(* Logix 5000 project; controller Comas_L4 vendor 1 type 14 code 193 rev 30.11; software revision 30.02; part 6 of 12 *)

        [6].Comas.Tete.Cam_Axe_Horizontal_Pan.C.x := 5.0, [6].Comas.Tete.Cam_Axe_Horizontal_Pan.C.y := 2.0, [6].Comas.Tete.Cam_Axe_Horizontal_Pan.D.x := 25.0, [6].Comas.Tete.Cam_Axe_Horizontal_Pan.D.y := 27.0, [6].Comas.Tete.Cam_Axe_Horizontal_Pan.E.x := 10.0, [6].Comas.Tete.Cam_Axe_Horizontal_Pan.E.y := 10.0, [6].Comas.Tete.Cam_Axe_Horizontal_Pan.F.x := 5.0, [6].Comas.Tete.Cam_Axe_Horizontal_Pan.G.x := 10.0, [6].Comas.Tete.Cam_Axe_Horizontal_Pan.G.y := -10.0, [6].Comas.Tete.Cam_Axe_Vertical_Pan.K.x := -10.0, [6].Comas.Tete.Cam_Axe_Vertical_Pan.L.x := -10.0, [6].Comas.Tete.Cam_Axe_Vertical_Pan.L.y := 12.0, [6].Comas.Tete.Cam_Axe_Vertical_Pan.M.x := 5.0, [6].Comas.Tete.Cam_Axe_Vertical_Pan.M.y := 5.0, [6].Comas.Tete.Cam_Axe_Vertical_Pan.N.x := 10.0, [6].Comas.Tete.Offset_Vertical_Droit := 45.0, [6].Comas.Tete.Offset_Horizontal_Droit := 95.0, [6].Comas.Tete.Reserve_Real1 := 3.0, [6].Comas.Pompe.Start_Cam_Logique_Avance := -9.0, [6].Comas.Pompe.Stop_Cam_Logique_Avance := 16.0, [6].Comas.Pompe.Start_Cam_Logique_Recul := 21.0, [6].Comas.Pompe.Stop_Cam_Logique_Recul := 33.0, [6].Comas.Pompe.Consigne_Vitesse_Avance := 19.6, [6].Comas.Pompe.Consigne_Acc_Dec_Avance := 40.0, [6].Comas.Pompe.Consigne_Jerk_Avance := 100.0, [6].Comas.Pompe.Consigne_Vitesse_Recul := -19.0, [6].Comas.Pompe.Consigne_Acc_Dec_Recul := 40.0, [6].Comas.Pompe.Consigne_Jerk_Recul := 100.0, [6].Comas.Pompe.Points_Pan.O.x := -15.0, [6].Comas.Pompe.Points_Pan.Q.x := 25.0, [6].Comas.Pompe.Points_Pan.U.x := 12.0, [6].Comas.Pompe.Reserve_Bool1 := 1, [6].Comas.Rouleaux.Syncho_Pompe := 1, [6].Comas.Rouleaux.Consigne_Vitesse := 25.0, [6].Comas.Rouleaux.Consigne_Acc_Dec := 40.0, [6].Comas.Rouleaux.Consigne_Jerk := 100.0, [6].Comas.Coupe_Fil.Start_Cam_Logique_Virtuelle := 11.0, [6].Comas.Coupe_Fil.Stop_Cam_Logique_Virtuelle := 21.0, [6].Comas.Coupe_Fil.Consigne_Vitesse_Virtuelle := 200.0, [6].Comas.Coupe_Fil.Consigne_Acc_Dec_Virtuelle := 1000.0, [6].Comas.Coupe_Fil.Consigne_Jerk_Virtuelle := 50.0, [6].Comas.Coupe_Fil.Cam_Axe[0].SegmentType := 1, [6].Comas.Coupe_Fil.Cam_Axe[1].Master := 180.0, [6].Comas.Coupe_Fil.Cam_Axe[1].Slave := 90.0, [6].Comas.Coupe_Fil.Cam_Axe[2].Master := 360.0, [6].Comas.Coupe_Fil.Cam_Axe[2].Slave := 360.0, [6].Comas.Coupe_Fil.Cam_Axe[2].SegmentType := 1, [6].Comas.Coupe_Fil.Points_Pan.W.x := 30.0, [6].Comas.Consigne_Vitesse_Manu_mm := 4.0, [6].Comas.Consigne_Acc_Decc_Manu_mm := 10.0, [6].Comas.Consigne_Jerk_Manu := 100.0, [6].Comas.Activation_Cam_Auto := 1, [6].Comas.Distance_CPT_Presence_Produit := 520, [6].Comas.Consigne_Vitesse_Manu_Tour := 10.0, [6].Comas.Consigne_Acc_Decc_Manu_Tour := 10.0, [6].Comas.Mode_Decoreuse_Cam_Logique := 1, [6].Comas.Reserve_Real3 := 1.0, [6].Comas.Reserve_Real4 := 1.0, [6].Comas.Reserve_Real5 := 5.0, [6].Comas.Reserve_Real6 := 200.0,
        [6].Reserve_Real2 := 200.0, [6].Reserve_Real3 := 10.0, [7].Name := 'SABLON 62x34 314SAB002', [7].Comas.Pas_Machine := 90, [7].Comas.Came_Maitre[1].Master := 90.0, [7].Comas.Came_Maitre[1].Slave := 90.0, [7].Comas.Longueur_Came_Maitre := 2, [7].Comas.Tete.Stop_Cam_Logique_Degagement := 10.0, [7].Comas.Tete.Position_Degagement_H := 50.0, [7].Comas.Tete.Position_Degagement_V := 35.0, [7].Comas.Tete.Hauteur_Tete := -6, [7].Comas.Tete.Cam_Axe_Horizontal[1].Master := 1.0, [7].Comas.Tete.Cam_Axe_Horizontal[1].SegmentType := 1, [7].Comas.Tete.Cam_Axe_Horizontal[2].Master := 6.0, [7].Comas.Tete.Cam_Axe_Horizontal[2].Slave := 5.0, [7].Comas.Tete.Cam_Axe_Horizontal[3].Master := 36.0, [7].Comas.Tete.Cam_Axe_Horizontal[3].Slave := 77.0, [7].Comas.Tete.Cam_Axe_Horizontal[3].SegmentType := 1, [7].Comas.Tete.Cam_Axe_Horizontal[4].Master := 46.0, [7].Comas.Tete.Cam_Axe_Horizontal[4].Slave := 87.0, [7].Comas.Tete.Cam_Axe_Horizontal[5].Master := 51.0, [7].Comas.Tete.Cam_Axe_Horizontal[5].Slave := 87.0, [7].Comas.Tete.Cam_Axe_Horizontal[5].SegmentType := 1, [7].Comas.Tete.Cam_Axe_Horizontal[6].Master := 61.0, [7].Comas.Tete.Cam_Axe_Horizontal[6].Slave := 77.0, [7].Comas.Tete.Cam_Axe_Horizontal[6].SegmentType := 1, [7].Comas.Tete.Cam_Axe_Horizontal[7].Master := 90.0, [7].Comas.Tete.Cam_Axe_Vertical[0].Slave := 15.0, [7].Comas.Tete.Cam_Axe_Vertical[1].Master := 1.0, [7].Comas.Tete.Cam_Axe_Vertical[1].Slave := 15.0, [7].Comas.Tete.Cam_Axe_Vertical[2].Master := 6.0, [7].Comas.Tete.Cam_Axe_Vertical[2].Slave := 15.0, [7].Comas.Tete.Cam_Axe_Vertical[3].Master := 48.0, [7].Comas.Tete.Cam_Axe_Vertical[3].Slave := 15.0, [7].Comas.Tete.Cam_Axe_Vertical[3].SegmentType := 1, [7].Comas.Tete.Cam_Axe_Vertical[4].Master := 58.0, [7].Comas.Tete.Cam_Axe_Vertical[4].Slave := 25.0, [7].Comas.Tete.Cam_Axe_Vertical[5].Master := 63.0, [7].Comas.Tete.Cam_Axe_Vertical[5].Slave := 25.0, [7].Comas.Tete.Cam_Axe_Vertical[5].SegmentType := 1, [7].Comas.Tete.Cam_Axe_Vertical[6].Master := 81.0, [7].Comas.Tete.Cam_Axe_Vertical[6].Slave := 15.0, [7].Comas.Tete.Cam_Axe_Vertical[7].Master := 90.0, [7].Comas.Tete.Cam_Axe_Vertical[7].Slave := 15.0, [7].Comas.Tete.Longueur_Cam_Axe_H := 8, [7].Comas.Tete.Offset_Vertical_Gauche := 38.0, [7].Comas.Tete.Offset_Horizontal_Gauche := 95.0, [7].Comas.Tete.Cam_Axe_Horizontal_Pan.B.x := 1.0, [7].Comas.Tete.Cam_Axe_Horizontal_Pan.C.x := 5.0, [7].Comas.Tete.Cam_Axe_Horizontal_Pan.C.y := 5.0, [7].Comas.Tete.Cam_Axe_Horizontal_Pan.D.x := 30.0, [7].Comas.Tete.Cam_Axe_Horizontal_Pan.D.y := 75.0, [7].Comas.Tete.Cam_Axe_Horizontal_Pan.E.x := 10.0, [7].Comas.Tete.Cam_Axe_Horizontal_Pan.E.y := 10.0, [7].Comas.Tete.Cam_Axe_Horizontal_Pan.F.x := 5.0, [7].Comas.Tete.Cam_Axe_Horizontal_Pan.G.x := 10.0, [7].Comas.Tete.Cam_Axe_Horizontal_Pan.G.y := -10.0, [7].Comas.Tete.Cam_Axe_Vertical_Pan.H.y := 15.0, [7].Comas.Tete.Cam_Axe_Vertical_Pan.I.y := 15.0, [7].Comas.Tete.Cam_Axe_Vertical_Pan.J.y := 15.0,
        [7].Comas.Tete.Cam_Axe_Vertical_Pan.K.x := 12.0, [7].Comas.Tete.Cam_Axe_Vertical_Pan.K.y := 15.0, [7].Comas.Tete.Cam_Axe_Vertical_Pan.L.x := 12.0, [7].Comas.Tete.Cam_Axe_Vertical_Pan.L.y := 25.0, [7].Comas.Tete.Cam_Axe_Vertical_Pan.M.x := 12.0, [7].Comas.Tete.Cam_Axe_Vertical_Pan.M.y := 25.0, [7].Comas.Tete.Cam_Axe_Vertical_Pan.N.x := 20.0, [7].Comas.Tete.Cam_Axe_Vertical_Pan.N.y := 15.0, [7].Comas.Tete.Offset_Vertical_Droit := 45.0, [7].Comas.Tete.Offset_Horizontal_Droit := 95.0, [7].Comas.Tete.Reserve_Real1 := -3.0, [7].Comas.Pompe.Start_Cam_Logique_Avance := -19.0, [7].Comas.Pompe.Stop_Cam_Logique_Avance := 31.0, [7].Comas.Pompe.Start_Cam_Logique_Recul := 43.0, [7].Comas.Pompe.Stop_Cam_Logique_Recul := 63.0, [7].Comas.Pompe.Consigne_Vitesse_Avance := 10.5, [7].Comas.Pompe.Consigne_Acc_Dec_Avance := 40.0, [7].Comas.Pompe.Consigne_Jerk_Avance := 100.0, [7].Comas.Pompe.Consigne_Vitesse_Recul := -10.0, [7].Comas.Pompe.Consigne_Acc_Dec_Recul := 40.0, [7].Comas.Pompe.Consigne_Jerk_Recul := 100.0, [7].Comas.Pompe.Points_Pan.O.x := -25.0, [7].Comas.Pompe.Points_Pan.Q.x := 50.0, [7].Comas.Pompe.Points_Pan.S.x := -5.0, [7].Comas.Pompe.Points_Pan.U.x := 20.0, [7].Comas.Pompe.Reserve_Bool1 := 1, [7].Comas.Rouleaux.Syncho_Pompe := 1, [7].Comas.Rouleaux.Consigne_Vitesse := 25.0, [7].Comas.Rouleaux.Consigne_Acc_Dec := 40.0, [7].Comas.Rouleaux.Consigne_Jerk := 100.0, [7].Comas.Coupe_Fil.Start_Cam_Logique_Virtuelle := 11.0, [7].Comas.Coupe_Fil.Stop_Cam_Logique_Virtuelle := 21.0, [7].Comas.Coupe_Fil.Consigne_Vitesse_Virtuelle := 200.0, [7].Comas.Coupe_Fil.Consigne_Acc_Dec_Virtuelle := 1000.0, [7].Comas.Coupe_Fil.Consigne_Jerk_Virtuelle := 50.0, [7].Comas.Coupe_Fil.Cam_Axe[0].SegmentType := 1, [7].Comas.Coupe_Fil.Cam_Axe[1].Master := 180.0, [7].Comas.Coupe_Fil.Cam_Axe[1].Slave := 90.0, [7].Comas.Coupe_Fil.Cam_Axe[2].Master := 360.0, [7].Comas.Coupe_Fil.Cam_Axe[2].Slave := 360.0, [7].Comas.Coupe_Fil.Cam_Axe[2].SegmentType := 1, [7].Comas.Coupe_Fil.Points_Pan.W.x := 30.0, [7].Comas.Consigne_Vitesse_Manu_mm := 2.0, [7].Comas.Consigne_Acc_Decc_Manu_mm := 10.0, [7].Comas.Consigne_Jerk_Manu := 100.0, [7].Comas.Activation_Cam_Auto := 1, [7].Comas.Distance_CPT_Presence_Produit := 520, [7].Comas.Consigne_Vitesse_Manu_Tour := 10.0, [7].Comas.Consigne_Acc_Decc_Manu_Tour := 10.0, [7].Comas.Mode_Decoreuse_Cam_Logique := 1, [7].Comas.Reserve_Real6 := 200.0, [8].Name := 'PALET CITRON 62X34', [8].Comas.Pas_Machine := 90, [8].Comas.Came_Maitre[1].Master := 90.0, [8].Comas.Came_Maitre[1].Slave := 90.0, [8].Comas.Longueur_Came_Maitre := 2, [8].Comas.Tete.Stop_Cam_Logique_Degagement := 10.0, [8].Comas.Tete.Position_Degagement_H := 50.0, [8].Comas.Tete.Position_Degagement_V := 35.0, [8].Comas.Tete.Hauteur_Tete := -2,
        [8].Comas.Tete.Cam_Axe_Horizontal[1].Master := 1.0, [8].Comas.Tete.Cam_Axe_Horizontal[1].SegmentType := 1, [8].Comas.Tete.Cam_Axe_Horizontal[2].Master := 6.0, [8].Comas.Tete.Cam_Axe_Horizontal[2].Slave := 5.0, [8].Comas.Tete.Cam_Axe_Horizontal[3].Master := 36.0, [8].Comas.Tete.Cam_Axe_Horizontal[3].Slave := 83.0, [8].Comas.Tete.Cam_Axe_Horizontal[3].SegmentType := 1, [8].Comas.Tete.Cam_Axe_Horizontal[4].Master := 46.0, [8].Comas.Tete.Cam_Axe_Horizontal[4].Slave := 93.0, [8].Comas.Tete.Cam_Axe_Horizontal[5].Master := 51.0, [8].Comas.Tete.Cam_Axe_Horizontal[5].Slave := 93.0, [8].Comas.Tete.Cam_Axe_Horizontal[5].SegmentType := 1, [8].Comas.Tete.Cam_Axe_Horizontal[6].Master := 61.0, [8].Comas.Tete.Cam_Axe_Horizontal[6].Slave := 83.0, [8].Comas.Tete.Cam_Axe_Horizontal[6].SegmentType := 1, [8].Comas.Tete.Cam_Axe_Horizontal[7].Master := 90.0, [8].Comas.Tete.Cam_Axe_Vertical[0].Slave := 15.0, [8].Comas.Tete.Cam_Axe_Vertical[1].Master := 1.0, [8].Comas.Tete.Cam_Axe_Vertical[1].Slave := 15.0, [8].Comas.Tete.Cam_Axe_Vertical[2].Master := 6.0, [8].Comas.Tete.Cam_Axe_Vertical[2].Slave := 15.0, [8].Comas.Tete.Cam_Axe_Vertical[3].Master := 46.0, [8].Comas.Tete.Cam_Axe_Vertical[3].Slave := 15.0, [8].Comas.Tete.Cam_Axe_Vertical[3].SegmentType := 1, [8].Comas.Tete.Cam_Axe_Vertical[4].Master := 56.0, [8].Comas.Tete.Cam_Axe_Vertical[4].Slave := 20.0, [8].Comas.Tete.Cam_Axe_Vertical[5].Master := 66.0, [8].Comas.Tete.Cam_Axe_Vertical[5].Slave := 20.0, [8].Comas.Tete.Cam_Axe_Vertical[5].SegmentType := 1, [8].Comas.Tete.Cam_Axe_Vertical[6].Master := 81.0, [8].Comas.Tete.Cam_Axe_Vertical[6].Slave := 15.0, [8].Comas.Tete.Cam_Axe_Vertical[7].Master := 90.0, [8].Comas.Tete.Cam_Axe_Vertical[7].Slave := 15.0, [8].Comas.Tete.Longueur_Cam_Axe_H := 8, [8].Comas.Tete.Offset_Vertical_Gauche := 38.0, [8].Comas.Tete.Offset_Horizontal_Gauche := 95.0, [8].Comas.Tete.Cam_Axe_Horizontal_Pan.B.x := 1.0, [8].Comas.Tete.Cam_Axe_Horizontal_Pan.C.x := 5.0, [8].Comas.Tete.Cam_Axe_Horizontal_Pan.C.y := 5.0, [8].Comas.Tete.Cam_Axe_Horizontal_Pan.D.x := 30.0, [8].Comas.Tete.Cam_Axe_Horizontal_Pan.D.y := 79.0, [8].Comas.Tete.Cam_Axe_Horizontal_Pan.E.x := 10.0, [8].Comas.Tete.Cam_Axe_Horizontal_Pan.E.y := 10.0, [8].Comas.Tete.Cam_Axe_Horizontal_Pan.F.x := 5.0, [8].Comas.Tete.Cam_Axe_Horizontal_Pan.G.x := 10.0, [8].Comas.Tete.Cam_Axe_Horizontal_Pan.G.y := -10.0, [8].Comas.Tete.Cam_Axe_Vertical_Pan.H.y := 15.0, [8].Comas.Tete.Cam_Axe_Vertical_Pan.I.y := 15.0, [8].Comas.Tete.Cam_Axe_Vertical_Pan.J.y := 15.0, [8].Comas.Tete.Cam_Axe_Vertical_Pan.K.x := 10.0, [8].Comas.Tete.Cam_Axe_Vertical_Pan.K.y := 15.0, [8].Comas.Tete.Cam_Axe_Vertical_Pan.L.x := 10.0, [8].Comas.Tete.Cam_Axe_Vertical_Pan.L.y := 20.0, [8].Comas.Tete.Cam_Axe_Vertical_Pan.M.x := 15.0, [8].Comas.Tete.Cam_Axe_Vertical_Pan.M.y := 20.0, [8].Comas.Tete.Cam_Axe_Vertical_Pan.N.x := 20.0, [8].Comas.Tete.Cam_Axe_Vertical_Pan.N.y := 15.0, [8].Comas.Tete.Offset_Vertical_Droit := 45.0, [8].Comas.Tete.Offset_Horizontal_Droit := 95.0, [8].Comas.Tete.Reserve_Real1 := -1.0,
        [8].Comas.Pompe.Start_Cam_Logique_Avance := -21.0, [8].Comas.Pompe.Stop_Cam_Logique_Avance := 25.0, [8].Comas.Pompe.Start_Cam_Logique_Recul := 26.0, [8].Comas.Pompe.Stop_Cam_Logique_Recul := 46.0, [8].Comas.Pompe.Consigne_Vitesse_Avance := 9.65, [8].Comas.Pompe.Consigne_Acc_Dec_Avance := 40.0, [8].Comas.Pompe.Consigne_Jerk_Avance := 100.0, [8].Comas.Pompe.Consigne_Vitesse_Recul := -10.0, [8].Comas.Pompe.Consigne_Acc_Dec_Recul := 40.0, [8].Comas.Pompe.Consigne_Jerk_Recul := 100.0, [8].Comas.Pompe.Points_Pan.O.x := -27.0, [8].Comas.Pompe.Points_Pan.Q.x := 46.0, [8].Comas.Pompe.Points_Pan.S.x := -20.0, [8].Comas.Pompe.Points_Pan.U.x := 20.0, [8].Comas.Pompe.Reserve_Bool1 := 1, [8].Comas.Rouleaux.Syncho_Pompe := 1, [8].Comas.Rouleaux.Consigne_Vitesse := 25.0, [8].Comas.Rouleaux.Consigne_Acc_Dec := 40.0, [8].Comas.Rouleaux.Consigne_Jerk := 100.0, [8].Comas.Coupe_Fil.Start_Cam_Logique_Virtuelle := 11.0, [8].Comas.Coupe_Fil.Stop_Cam_Logique_Virtuelle := 21.0, [8].Comas.Coupe_Fil.Consigne_Vitesse_Virtuelle := 200.0, [8].Comas.Coupe_Fil.Consigne_Acc_Dec_Virtuelle := 1000.0, [8].Comas.Coupe_Fil.Consigne_Jerk_Virtuelle := 50.0, [8].Comas.Coupe_Fil.Cam_Axe[0].SegmentType := 1, [8].Comas.Coupe_Fil.Cam_Axe[1].Master := 180.0, [8].Comas.Coupe_Fil.Cam_Axe[1].Slave := 90.0, [8].Comas.Coupe_Fil.Cam_Axe[2].Master := 360.0, [8].Comas.Coupe_Fil.Cam_Axe[2].Slave := 360.0, [8].Comas.Coupe_Fil.Cam_Axe[2].SegmentType := 1, [8].Comas.Coupe_Fil.Points_Pan.W.x := 30.0, [8].Comas.Consigne_Vitesse_Manu_mm := 4.0, [8].Comas.Consigne_Acc_Decc_Manu_mm := 10.0, [8].Comas.Consigne_Jerk_Manu := 100.0, [8].Comas.Activation_Cam_Auto := 1, [8].Comas.Distance_CPT_Presence_Produit := 520, [8].Comas.Consigne_Vitesse_Manu_Tour := 10.0, [8].Comas.Consigne_Acc_Decc_Manu_Tour := 10.0, [8].Comas.Mode_Decoreuse_Cam_Logique := 1, [8].Comas.Reserve_Real6 := 200.0, [9].Name := 'LISON', [9].Comas.Pas_Machine := 70, [9].Comas.Came_Maitre[1].Master := 70.0, [9].Comas.Came_Maitre[1].Slave := 70.0, [9].Comas.Longueur_Came_Maitre := 2, [9].Comas.Tete.Stop_Cam_Logique_Degagement := 10.0, [9].Comas.Tete.Position_Degagement_H := 50.0, [9].Comas.Tete.Position_Degagement_V := 35.0, [9].Comas.Tete.Hauteur_Tete := -3, [9].Comas.Tete.Cam_Axe_Horizontal[1].Master := 1.0, [9].Comas.Tete.Cam_Axe_Horizontal[1].SegmentType := 1, [9].Comas.Tete.Cam_Axe_Horizontal[2].Master := 6.0, [9].Comas.Tete.Cam_Axe_Horizontal[2].Slave := 5.0, [9].Comas.Tete.Cam_Axe_Horizontal[2].SegmentType := 1, [9].Comas.Tete.Cam_Axe_Horizontal[3].Master := 31.0, [9].Comas.Tete.Cam_Axe_Horizontal[3].Slave := 32.0, [9].Comas.Tete.Cam_Axe_Horizontal[3].SegmentType := 1, [9].Comas.Tete.Cam_Axe_Horizontal[4].Master := 41.0, [9].Comas.Tete.Cam_Axe_Horizontal[4].Slave := 37.0, [9].Comas.Tete.Cam_Axe_Horizontal[5].Master := 46.0,
        [9].Comas.Tete.Cam_Axe_Horizontal[5].Slave := 37.0, [9].Comas.Tete.Cam_Axe_Horizontal[5].SegmentType := 1, [9].Comas.Tete.Cam_Axe_Horizontal[6].Master := 56.0, [9].Comas.Tete.Cam_Axe_Horizontal[6].Slave := 27.0, [9].Comas.Tete.Cam_Axe_Horizontal[6].SegmentType := 1, [9].Comas.Tete.Cam_Axe_Horizontal[7].Master := 70.0, [9].Comas.Tete.Cam_Axe_Vertical[1].Master := 1.0, [9].Comas.Tete.Cam_Axe_Vertical[2].Master := 6.0, [9].Comas.Tete.Cam_Axe_Vertical[3].Master := 21.0, [9].Comas.Tete.Cam_Axe_Vertical[3].SegmentType := 1, [9].Comas.Tete.Cam_Axe_Vertical[4].Master := 31.0, [9].Comas.Tete.Cam_Axe_Vertical[4].Slave := 6.0, [9].Comas.Tete.Cam_Axe_Vertical[5].Master := 51.0, [9].Comas.Tete.Cam_Axe_Vertical[5].Slave := 6.0, [9].Comas.Tete.Cam_Axe_Vertical[5].SegmentType := 1, [9].Comas.Tete.Cam_Axe_Vertical[6].Master := 66.0, [9].Comas.Tete.Cam_Axe_Vertical[6].Slave := 6.0, [9].Comas.Tete.Cam_Axe_Vertical[7].Master := 70.0, [9].Comas.Tete.Longueur_Cam_Axe_H := 8, [9].Comas.Tete.Offset_Vertical_Gauche := 38.0, [9].Comas.Tete.Offset_Horizontal_Gauche := 95.0, [9].Comas.Tete.Cam_Axe_Horizontal_Pan.B.x := 1.0, [9].Comas.Tete.Cam_Axe_Horizontal_Pan.C.x := 5.0, [9].Comas.Tete.Cam_Axe_Horizontal_Pan.C.y := 5.0, [9].Comas.Tete.Cam_Axe_Horizontal_Pan.D.x := 25.0, [9].Comas.Tete.Cam_Axe_Horizontal_Pan.D.y := 27.0, [9].Comas.Tete.Cam_Axe_Horizontal_Pan.E.x := 10.0, [9].Comas.Tete.Cam_Axe_Horizontal_Pan.E.y := 5.0, [9].Comas.Tete.Cam_Axe_Horizontal_Pan.F.x := 5.0, [9].Comas.Tete.Cam_Axe_Horizontal_Pan.G.x := 10.0, [9].Comas.Tete.Cam_Axe_Horizontal_Pan.G.y := -10.0, [9].Comas.Tete.Cam_Axe_Vertical_Pan.K.x := -10.0, [9].Comas.Tete.Cam_Axe_Vertical_Pan.L.x := -10.0, [9].Comas.Tete.Cam_Axe_Vertical_Pan.L.y := 6.0, [9].Comas.Tete.Cam_Axe_Vertical_Pan.M.x := 5.0, [9].Comas.Tete.Cam_Axe_Vertical_Pan.M.y := 6.0, [9].Comas.Tete.Cam_Axe_Vertical_Pan.N.x := 10.0, [9].Comas.Tete.Cam_Axe_Vertical_Pan.N.y := 6.0, [9].Comas.Tete.Offset_Vertical_Droit := 45.0, [9].Comas.Tete.Offset_Horizontal_Droit := 95.0, [9].Comas.Pompe.Start_Cam_Logique_Avance := -9.0, [9].Comas.Pompe.Stop_Cam_Logique_Avance := 16.0, [9].Comas.Pompe.Start_Cam_Logique_Recul := 21.0, [9].Comas.Pompe.Stop_Cam_Logique_Recul := 33.0, [9].Comas.Pompe.Consigne_Vitesse_Avance := 15.6, [9].Comas.Pompe.Consigne_Acc_Dec_Avance := 40.0, [9].Comas.Pompe.Consigne_Jerk_Avance := 100.0, [9].Comas.Pompe.Consigne_Vitesse_Recul := -16.0, [9].Comas.Pompe.Consigne_Acc_Dec_Recul := 40.0, [9].Comas.Pompe.Consigne_Jerk_Recul := 100.0, [9].Comas.Pompe.Points_Pan.O.x := -15.0, [9].Comas.Pompe.Points_Pan.Q.x := 25.0, [9].Comas.Pompe.Points_Pan.U.x := 12.0, [9].Comas.Pompe.Reserve_Bool1 := 1, [9].Comas.Rouleaux.Syncho_Pompe := 1, [9].Comas.Rouleaux.Consigne_Vitesse := 25.0, [9].Comas.Rouleaux.Consigne_Acc_Dec := 40.0, [9].Comas.Rouleaux.Consigne_Jerk := 100.0, [9].Comas.Coupe_Fil.Start_Cam_Logique_Virtuelle := 11.0, [9].Comas.Coupe_Fil.Stop_Cam_Logique_Virtuelle := 21.0,
        [9].Comas.Coupe_Fil.Consigne_Vitesse_Virtuelle := 200.0, [9].Comas.Coupe_Fil.Consigne_Acc_Dec_Virtuelle := 1000.0, [9].Comas.Coupe_Fil.Consigne_Jerk_Virtuelle := 50.0, [9].Comas.Coupe_Fil.Cam_Axe[0].SegmentType := 1, [9].Comas.Coupe_Fil.Cam_Axe[1].Master := 180.0, [9].Comas.Coupe_Fil.Cam_Axe[1].Slave := 90.0, [9].Comas.Coupe_Fil.Cam_Axe[2].Master := 360.0, [9].Comas.Coupe_Fil.Cam_Axe[2].Slave := 360.0, [9].Comas.Coupe_Fil.Cam_Axe[2].SegmentType := 1, [9].Comas.Coupe_Fil.Points_Pan.W.x := 30.0, [9].Comas.Consigne_Vitesse_Manu_mm := 4.0, [9].Comas.Consigne_Acc_Decc_Manu_mm := 10.0, [9].Comas.Consigne_Jerk_Manu := 100.0, [9].Comas.Activation_Cam_Auto := 1, [9].Comas.Distance_CPT_Presence_Produit := 520, [9].Comas.Consigne_Vitesse_Manu_Tour := 10.0, [9].Comas.Consigne_Acc_Decc_Manu_Tour := 10.0, [9].Comas.Mode_Decoreuse_Cam_Logique := 1, [9].Comas.Reserve_Real3 := 1.0, [9].Comas.Reserve_Real4 := 1.0, [9].Comas.Reserve_Real5 := 5.0, [9].Comas.Reserve_Real6 := 200.0, [9].Reserve_Real2 := 200.0, [9].Reserve_Real3 := 10.0, [10].Name := 'PAL CISSP 62x34 318PJL005', [10].Comas.Pas_Machine := 90, [10].Comas.Came_Maitre[1].Master := 90.0, [10].Comas.Came_Maitre[1].Slave := 90.0, [10].Comas.Longueur_Came_Maitre := 2, [10].Comas.Tete.Stop_Cam_Logique_Degagement := 10.0, [10].Comas.Tete.Position_Degagement_H := 50.0, [10].Comas.Tete.Position_Degagement_V := 35.0, [10].Comas.Tete.Hauteur_Tete := -14, [10].Comas.Tete.Cam_Axe_Horizontal[1].Master := 1.0, [10].Comas.Tete.Cam_Axe_Horizontal[1].SegmentType := 1, [10].Comas.Tete.Cam_Axe_Horizontal[2].Master := 6.0, [10].Comas.Tete.Cam_Axe_Horizontal[2].Slave := 5.0, [10].Comas.Tete.Cam_Axe_Horizontal[3].Master := 36.0, [10].Comas.Tete.Cam_Axe_Horizontal[3].Slave := 79.0, [10].Comas.Tete.Cam_Axe_Horizontal[3].SegmentType := 1, [10].Comas.Tete.Cam_Axe_Horizontal[4].Master := 46.0, [10].Comas.Tete.Cam_Axe_Horizontal[4].Slave := 89.0, [10].Comas.Tete.Cam_Axe_Horizontal[5].Master := 51.0, [10].Comas.Tete.Cam_Axe_Horizontal[5].Slave := 89.0, [10].Comas.Tete.Cam_Axe_Horizontal[5].SegmentType := 1, [10].Comas.Tete.Cam_Axe_Horizontal[6].Master := 61.0, [10].Comas.Tete.Cam_Axe_Horizontal[6].Slave := 79.0, [10].Comas.Tete.Cam_Axe_Horizontal[6].SegmentType := 1, [10].Comas.Tete.Cam_Axe_Horizontal[7].Master := 90.0, [10].Comas.Tete.Cam_Axe_Vertical[0].Slave := 15.0, [10].Comas.Tete.Cam_Axe_Vertical[1].Master := 1.0, [10].Comas.Tete.Cam_Axe_Vertical[1].Slave := 15.0, [10].Comas.Tete.Cam_Axe_Vertical[2].Master := 6.0, [10].Comas.Tete.Cam_Axe_Vertical[2].Slave := 15.0, [10].Comas.Tete.Cam_Axe_Vertical[3].Master := 46.0, [10].Comas.Tete.Cam_Axe_Vertical[3].Slave := 15.0, [10].Comas.Tete.Cam_Axe_Vertical[3].SegmentType := 1, [10].Comas.Tete.Cam_Axe_Vertical[4].Master := 56.0, [10].Comas.Tete.Cam_Axe_Vertical[4].Slave := 20.0, [10].Comas.Tete.Cam_Axe_Vertical[5].Master := 66.0,
        [10].Comas.Tete.Cam_Axe_Vertical[5].Slave := 20.0, [10].Comas.Tete.Cam_Axe_Vertical[5].SegmentType := 1, [10].Comas.Tete.Cam_Axe_Vertical[6].Master := 81.0, [10].Comas.Tete.Cam_Axe_Vertical[6].Slave := 15.0, [10].Comas.Tete.Cam_Axe_Vertical[7].Master := 90.0, [10].Comas.Tete.Cam_Axe_Vertical[7].Slave := 15.0, [10].Comas.Tete.Longueur_Cam_Axe_H := 8, [10].Comas.Tete.Offset_Vertical_Gauche := 38.0, [10].Comas.Tete.Offset_Horizontal_Gauche := 95.0, [10].Comas.Tete.Cam_Axe_Horizontal_Pan.B.x := 1.0, [10].Comas.Tete.Cam_Axe_Horizontal_Pan.C.x := 5.0, [10].Comas.Tete.Cam_Axe_Horizontal_Pan.C.y := 5.0, [10].Comas.Tete.Cam_Axe_Horizontal_Pan.D.x := 30.0, [10].Comas.Tete.Cam_Axe_Horizontal_Pan.D.y := 79.0, [10].Comas.Tete.Cam_Axe_Horizontal_Pan.E.x := 10.0, [10].Comas.Tete.Cam_Axe_Horizontal_Pan.E.y := 10.0, [10].Comas.Tete.Cam_Axe_Horizontal_Pan.F.x := 5.0, [10].Comas.Tete.Cam_Axe_Horizontal_Pan.G.x := 10.0, [10].Comas.Tete.Cam_Axe_Horizontal_Pan.G.y := -10.0, [10].Comas.Tete.Cam_Axe_Vertical_Pan.H.y := 15.0, [10].Comas.Tete.Cam_Axe_Vertical_Pan.I.y := 15.0, [10].Comas.Tete.Cam_Axe_Vertical_Pan.J.y := 15.0, [10].Comas.Tete.Cam_Axe_Vertical_Pan.K.x := 10.0, [10].Comas.Tete.Cam_Axe_Vertical_Pan.K.y := 15.0, [10].Comas.Tete.Cam_Axe_Vertical_Pan.L.x := 10.0, [10].Comas.Tete.Cam_Axe_Vertical_Pan.L.y := 20.0, [10].Comas.Tete.Cam_Axe_Vertical_Pan.M.x := 15.0, [10].Comas.Tete.Cam_Axe_Vertical_Pan.M.y := 20.0, [10].Comas.Tete.Cam_Axe_Vertical_Pan.N.x := 20.0, [10].Comas.Tete.Cam_Axe_Vertical_Pan.N.y := 15.0, [10].Comas.Tete.Offset_Vertical_Droit := 45.0, [10].Comas.Tete.Offset_Horizontal_Droit := 95.0, [10].Comas.Tete.Reserve_Real1 := -5.0, [10].Comas.Pompe.Start_Cam_Logique_Avance := -13.0, [10].Comas.Pompe.Stop_Cam_Logique_Avance := 33.0, [10].Comas.Pompe.Start_Cam_Logique_Recul := 26.0, [10].Comas.Pompe.Stop_Cam_Logique_Recul := 46.0, [10].Comas.Pompe.Consigne_Vitesse_Avance := 11.8, [10].Comas.Pompe.Consigne_Acc_Dec_Avance := 40.0, [10].Comas.Pompe.Consigne_Jerk_Avance := 100.0, [10].Comas.Pompe.Consigne_Vitesse_Recul := -12.0, [10].Comas.Pompe.Consigne_Acc_Dec_Recul := 40.0, [10].Comas.Pompe.Consigne_Jerk_Recul := 100.0, [10].Comas.Pompe.Points_Pan.O.x := -19.0, [10].Comas.Pompe.Points_Pan.Q.x := 46.0, [10].Comas.Pompe.Points_Pan.S.x := -20.0, [10].Comas.Pompe.Points_Pan.U.x := 20.0, [10].Comas.Pompe.Reserve_Bool1 := 1, [10].Comas.Rouleaux.Syncho_Pompe := 1, [10].Comas.Rouleaux.Consigne_Vitesse := 20.0, [10].Comas.Rouleaux.Consigne_Acc_Dec := 40.0, [10].Comas.Rouleaux.Consigne_Jerk := 100.0, [10].Comas.Coupe_Fil.Start_Cam_Logique_Virtuelle := 11.0, [10].Comas.Coupe_Fil.Stop_Cam_Logique_Virtuelle := 21.0, [10].Comas.Coupe_Fil.Consigne_Vitesse_Virtuelle := 200.0, [10].Comas.Coupe_Fil.Consigne_Acc_Dec_Virtuelle := 1000.0, [10].Comas.Coupe_Fil.Consigne_Jerk_Virtuelle := 50.0, [10].Comas.Coupe_Fil.Cam_Axe[0].SegmentType := 1, [10].Comas.Coupe_Fil.Cam_Axe[1].Master := 180.0, [10].Comas.Coupe_Fil.Cam_Axe[1].Slave := 90.0,
        [10].Comas.Coupe_Fil.Cam_Axe[2].Master := 360.0, [10].Comas.Coupe_Fil.Cam_Axe[2].Slave := 360.0, [10].Comas.Coupe_Fil.Cam_Axe[2].SegmentType := 1, [10].Comas.Coupe_Fil.Points_Pan.W.x := 30.0, [10].Comas.Consigne_Vitesse_Manu_mm := 4.0, [10].Comas.Consigne_Acc_Decc_Manu_mm := 10.0, [10].Comas.Consigne_Jerk_Manu := 100.0, [10].Comas.Activation_Cam_Auto := 1, [10].Comas.Distance_CPT_Presence_Produit := 520, [10].Comas.Consigne_Vitesse_Manu_Tour := 10.0, [10].Comas.Consigne_Acc_Decc_Manu_Tour := 10.0, [10].Comas.Mode_Decoreuse_Cam_Logique := 1, [10].Comas.Reserve_Real3 := 1.0, [10].Comas.Reserve_Real4 := 1.0, [10].Comas.Reserve_Real5 := 5.0, [10].Comas.Reserve_Real6 := 200.0, [10].Reserve_Real2 := 200.0, [10].Reserve_Real3 := 10.0, [11].Name := 'palet MDLZ', [11].Comas.Pas_Machine := 60, [11].Comas.Came_Maitre[1].Master := 60.0, [11].Comas.Came_Maitre[1].Slave := 60.0, [11].Comas.Longueur_Came_Maitre := 2, [11].Comas.Tete.Stop_Cam_Logique_Degagement := 10.0, [11].Comas.Tete.Position_Degagement_H := 50.0, [11].Comas.Tete.Position_Degagement_V := 35.0, [11].Comas.Tete.Hauteur_Tete := -9, [11].Comas.Tete.Cam_Axe_Horizontal[1].Master := 1.0, [11].Comas.Tete.Cam_Axe_Horizontal[1].SegmentType := 1, [11].Comas.Tete.Cam_Axe_Horizontal[2].Master := 6.0, [11].Comas.Tete.Cam_Axe_Horizontal[2].Slave := 2.0, [11].Comas.Tete.Cam_Axe_Horizontal[3].Master := 21.0, [11].Comas.Tete.Cam_Axe_Horizontal[3].Slave := 24.0, [11].Comas.Tete.Cam_Axe_Horizontal[3].SegmentType := 1, [11].Comas.Tete.Cam_Axe_Horizontal[4].Master := 31.0, [11].Comas.Tete.Cam_Axe_Horizontal[4].Slave := 29.0, [11].Comas.Tete.Cam_Axe_Horizontal[5].Master := 36.0, [11].Comas.Tete.Cam_Axe_Horizontal[5].Slave := 29.0, [11].Comas.Tete.Cam_Axe_Horizontal[5].SegmentType := 1, [11].Comas.Tete.Cam_Axe_Horizontal[6].Master := 46.0, [11].Comas.Tete.Cam_Axe_Horizontal[6].Slave := 19.0, [11].Comas.Tete.Cam_Axe_Horizontal[6].SegmentType := 1, [11].Comas.Tete.Cam_Axe_Horizontal[7].Master := 60.0, [11].Comas.Tete.Cam_Axe_Vertical[1].Master := 1.0, [11].Comas.Tete.Cam_Axe_Vertical[2].Master := 6.0, [11].Comas.Tete.Cam_Axe_Vertical[3].Master := 11.0, [11].Comas.Tete.Cam_Axe_Vertical[3].SegmentType := 1, [11].Comas.Tete.Cam_Axe_Vertical[4].Master := 21.0, [11].Comas.Tete.Cam_Axe_Vertical[4].Slave := 3.0, [11].Comas.Tete.Cam_Axe_Vertical[5].Master := 41.0, [11].Comas.Tete.Cam_Axe_Vertical[5].Slave := 3.0, [11].Comas.Tete.Cam_Axe_Vertical[5].SegmentType := 1, [11].Comas.Tete.Cam_Axe_Vertical[6].Master := 56.0, [11].Comas.Tete.Cam_Axe_Vertical[7].Master := 60.0, [11].Comas.Tete.Longueur_Cam_Axe_H := 8, [11].Comas.Tete.Offset_Vertical_Gauche := 38.0, [11].Comas.Tete.Offset_Horizontal_Gauche := 95.0, [11].Comas.Tete.Cam_Axe_Horizontal_Pan.B.x := 1.0, [11].Comas.Tete.Cam_Axe_Horizontal_Pan.C.x := 5.0, [11].Comas.Tete.Cam_Axe_Horizontal_Pan.C.y := 2.0,
        [11].Comas.Tete.Cam_Axe_Horizontal_Pan.D.x := 15.0, [11].Comas.Tete.Cam_Axe_Horizontal_Pan.D.y := 25.0, [11].Comas.Tete.Cam_Axe_Horizontal_Pan.E.x := 10.0, [11].Comas.Tete.Cam_Axe_Horizontal_Pan.E.y := 5.0, [11].Comas.Tete.Cam_Axe_Horizontal_Pan.F.x := 5.0, [11].Comas.Tete.Cam_Axe_Horizontal_Pan.G.x := 10.0, [11].Comas.Tete.Cam_Axe_Horizontal_Pan.G.y := -10.0, [11].Comas.Tete.Cam_Axe_Vertical_Pan.K.x := -10.0, [11].Comas.Tete.Cam_Axe_Vertical_Pan.L.x := -10.0, [11].Comas.Tete.Cam_Axe_Vertical_Pan.L.y := 3.0, [11].Comas.Tete.Cam_Axe_Vertical_Pan.M.x := 5.0, [11].Comas.Tete.Cam_Axe_Vertical_Pan.M.y := 3.0, [11].Comas.Tete.Cam_Axe_Vertical_Pan.N.x := 10.0, [11].Comas.Tete.Offset_Vertical_Droit := 45.0, [11].Comas.Tete.Offset_Horizontal_Droit := 95.0, [11].Comas.Tete.Reserve_Real1 := -3.0, [11].Comas.Pompe.Start_Cam_Logique_Avance := -8.0, [11].Comas.Pompe.Stop_Cam_Logique_Avance := 7.0, [11].Comas.Pompe.Start_Cam_Logique_Recul := 7.0, [11].Comas.Pompe.Stop_Cam_Logique_Recul := 22.0, [11].Comas.Pompe.Consigne_Vitesse_Avance := 50.8, [11].Comas.Pompe.Consigne_Acc_Dec_Avance := 40.0, [11].Comas.Pompe.Consigne_Jerk_Avance := 100.0, [11].Comas.Pompe.Consigne_Vitesse_Recul := -28.0, [11].Comas.Pompe.Consigne_Acc_Dec_Recul := 40.0, [11].Comas.Pompe.Consigne_Jerk_Recul := 100.0, [11].Comas.Pompe.Points_Pan.O.x := -14.0, [11].Comas.Pompe.Points_Pan.Q.x := 15.0, [11].Comas.Pompe.Points_Pan.S.x := -4.0, [11].Comas.Pompe.Points_Pan.U.x := 15.0, [11].Comas.Pompe.Reserve_Bool1 := 1, [11].Comas.Rouleaux.Consigne_Vitesse := 25.0, [11].Comas.Rouleaux.Consigne_Acc_Dec := 40.0, [11].Comas.Rouleaux.Consigne_Jerk := 100.0, [11].Comas.Rouleaux.Reserve_Real1 := -15.0, [11].Comas.Coupe_Fil.Start_Cam_Logique_Virtuelle := 11.0, [11].Comas.Coupe_Fil.Stop_Cam_Logique_Virtuelle := 21.0, [11].Comas.Coupe_Fil.Consigne_Vitesse_Virtuelle := 200.0, [11].Comas.Coupe_Fil.Consigne_Acc_Dec_Virtuelle := 1000.0, [11].Comas.Coupe_Fil.Consigne_Jerk_Virtuelle := 50.0, [11].Comas.Coupe_Fil.Cam_Axe[0].SegmentType := 1, [11].Comas.Coupe_Fil.Cam_Axe[1].Master := 180.0, [11].Comas.Coupe_Fil.Cam_Axe[1].Slave := 90.0, [11].Comas.Coupe_Fil.Cam_Axe[2].Master := 360.0, [11].Comas.Coupe_Fil.Cam_Axe[2].Slave := 360.0, [11].Comas.Coupe_Fil.Cam_Axe[2].SegmentType := 1, [11].Comas.Coupe_Fil.Points_Pan.W.x := 30.0, [11].Comas.Consigne_Vitesse_Manu_mm := 4.0, [11].Comas.Consigne_Acc_Decc_Manu_mm := 10.0, [11].Comas.Consigne_Jerk_Manu := 100.0, [11].Comas.Activation_Cam_Auto := 1, [11].Comas.Distance_CPT_Presence_Produit := 520, [11].Comas.Consigne_Vitesse_Manu_Tour := 10.0, [11].Comas.Consigne_Acc_Decc_Manu_Tour := 10.0, [11].Comas.Mode_Decoreuse_Cam_Logique := 1, [11].Comas.Reserve_Real3 := 1.0, [11].Comas.Reserve_Real4 := 1.0, [11].Comas.Reserve_Real5 := 5.0, [11].Comas.Reserve_Real6 := 200.0, [11].Reserve_Real2 := 200.0,
        [11].Reserve_Real3 := 10.0, [12].Name := 'COOKIE 314MIN011', [12].Comas.Pas_Machine := 95, [12].Comas.Came_Maitre[1].Master := 95.0, [12].Comas.Came_Maitre[1].Slave := 95.0, [12].Comas.Longueur_Came_Maitre := 2, [12].Comas.Tete.Stop_Cam_Logique_Degagement := 10.0, [12].Comas.Tete.Position_Degagement_H := 50.0, [12].Comas.Tete.Position_Degagement_V := 35.0, [12].Comas.Tete.Hauteur_Tete := -1, [12].Comas.Tete.Cam_Axe_Horizontal[1].Master := 1.0, [12].Comas.Tete.Cam_Axe_Horizontal[1].SegmentType := 1, [12].Comas.Tete.Cam_Axe_Horizontal[2].Master := 11.0, [12].Comas.Tete.Cam_Axe_Horizontal[2].Slave := 5.0, [12].Comas.Tete.Cam_Axe_Horizontal[3].Master := 41.0, [12].Comas.Tete.Cam_Axe_Horizontal[3].Slave := 35.0, [12].Comas.Tete.Cam_Axe_Horizontal[3].SegmentType := 1, [12].Comas.Tete.Cam_Axe_Horizontal[4].Master := 51.0, [12].Comas.Tete.Cam_Axe_Horizontal[4].Slave := 40.0, [12].Comas.Tete.Cam_Axe_Horizontal[5].Master := 61.0, [12].Comas.Tete.Cam_Axe_Horizontal[5].Slave := 40.0, [12].Comas.Tete.Cam_Axe_Horizontal[5].SegmentType := 1, [12].Comas.Tete.Cam_Axe_Horizontal[6].Master := 71.0, [12].Comas.Tete.Cam_Axe_Horizontal[6].Slave := 30.0, [12].Comas.Tete.Cam_Axe_Horizontal[6].SegmentType := 1, [12].Comas.Tete.Cam_Axe_Horizontal[7].Master := 95.0, [12].Comas.Tete.Cam_Axe_Vertical[1].Master := 1.0, [12].Comas.Tete.Cam_Axe_Vertical[2].Master := 11.0, [12].Comas.Tete.Cam_Axe_Vertical[3].Master := 41.0, [12].Comas.Tete.Cam_Axe_Vertical[3].SegmentType := 1, [12].Comas.Tete.Cam_Axe_Vertical[4].Master := 56.0, [12].Comas.Tete.Cam_Axe_Vertical[4].Slave := 10.0, [12].Comas.Tete.Cam_Axe_Vertical[5].Master := 66.0, [12].Comas.Tete.Cam_Axe_Vertical[5].Slave := 10.0, [12].Comas.Tete.Cam_Axe_Vertical[5].SegmentType := 1, [12].Comas.Tete.Cam_Axe_Vertical[6].Master := 86.0, [12].Comas.Tete.Cam_Axe_Vertical[7].Master := 95.0, [12].Comas.Tete.Longueur_Cam_Axe_H := 8, [12].Comas.Tete.Offset_Vertical_Gauche := 38.0, [12].Comas.Tete.Offset_Horizontal_Gauche := 95.0, [12].Comas.Tete.Cam_Axe_Horizontal_Pan.B.x := 1.0, [12].Comas.Tete.Cam_Axe_Horizontal_Pan.C.x := 10.0, [12].Comas.Tete.Cam_Axe_Horizontal_Pan.C.y := 5.0, [12].Comas.Tete.Cam_Axe_Horizontal_Pan.D.x := 30.0, [12].Comas.Tete.Cam_Axe_Horizontal_Pan.D.y := 30.0, [12].Comas.Tete.Cam_Axe_Horizontal_Pan.E.x := 10.0, [12].Comas.Tete.Cam_Axe_Horizontal_Pan.E.y := 5.0, [12].Comas.Tete.Cam_Axe_Horizontal_Pan.F.x := 10.0, [12].Comas.Tete.Cam_Axe_Horizontal_Pan.G.x := 10.0, [12].Comas.Tete.Cam_Axe_Horizontal_Pan.G.y := -10.0, [12].Comas.Tete.Cam_Axe_Vertical_Pan.L.x := 5.0, [12].Comas.Tete.Cam_Axe_Vertical_Pan.L.y := 10.0, [12].Comas.Tete.Cam_Axe_Vertical_Pan.M.x := 5.0, [12].Comas.Tete.Cam_Axe_Vertical_Pan.M.y := 10.0, [12].Comas.Tete.Cam_Axe_Vertical_Pan.N.x := 15.0, [12].Comas.Tete.Offset_Vertical_Droit := 45.0, [12].Comas.Tete.Offset_Horizontal_Droit := 95.0, [12].Comas.Pompe.Start_Cam_Logique_Avance := 1.0, [12].Comas.Pompe.Stop_Cam_Logique_Avance := 14.0, [12].Comas.Pompe.Start_Cam_Logique_Recul := 16.0,
        [12].Comas.Pompe.Stop_Cam_Logique_Recul := 31.0, [12].Comas.Pompe.Consigne_Vitesse_Avance := 14.0, [12].Comas.Pompe.Consigne_Acc_Dec_Avance := 40.0, [12].Comas.Pompe.Consigne_Jerk_Avance := 100.0, [12].Comas.Pompe.Consigne_Acc_Dec_Recul := 40.0, [12].Comas.Pompe.Consigne_Jerk_Recul := 100.0, [12].Comas.Pompe.Points_Pan.O.x := -10.0, [12].Comas.Pompe.Points_Pan.Q.x := 13.0, [12].Comas.Pompe.Points_Pan.S.x := -25.0, [12].Comas.Pompe.Points_Pan.U.x := 15.0, [12].Comas.Pompe.Reserve_Bool1 := 1, [12].Comas.Rouleaux.Syncho_Pompe := 1, [12].Comas.Rouleaux.Consigne_Vitesse := 30.0, [12].Comas.Rouleaux.Consigne_Acc_Dec := 40.0, [12].Comas.Rouleaux.Consigne_Jerk := 100.0, [12].Comas.Rouleaux.Reserve_Real1 := -20.0, [12].Comas.Coupe_Fil.Activation := 1, [12].Comas.Coupe_Fil.Start_Cam_Logique_Virtuelle := 11.0, [12].Comas.Coupe_Fil.Stop_Cam_Logique_Virtuelle := 21.0, [12].Comas.Coupe_Fil.Consigne_Vitesse_Virtuelle := 250.0, [12].Comas.Coupe_Fil.Consigne_Acc_Dec_Virtuelle := 1000.0, [12].Comas.Coupe_Fil.Consigne_Jerk_Virtuelle := 50.0, [12].Comas.Coupe_Fil.Cam_Axe[0].SegmentType := 1, [12].Comas.Coupe_Fil.Cam_Axe[1].Master := 180.0, [12].Comas.Coupe_Fil.Cam_Axe[1].Slave := 180.0, [12].Comas.Coupe_Fil.Cam_Axe[2].Master := 250.0, [12].Comas.Coupe_Fil.Cam_Axe[2].Slave := 180.0, [12].Comas.Coupe_Fil.Cam_Axe[2].SegmentType := 1, [12].Comas.Coupe_Fil.Cam_Axe[3].Master := 360.0, [12].Comas.Coupe_Fil.Cam_Axe[3].Slave := 360.0, [12].Comas.Coupe_Fil.Cam_Axe[3].SegmentType := 1, [12].Comas.Coupe_Fil.Cam_Axe[4].SegmentType := 1, [12].Comas.Coupe_Fil.Points_Pan.W.x := -40.0, [12].Comas.Coupe_Fil.Reserve_Bool1 := 1, [12].Comas.Consigne_Vitesse_Manu_mm := 2.0, [12].Comas.Consigne_Acc_Decc_Manu_mm := 10.0, [12].Comas.Consigne_Jerk_Manu := 100.0, [12].Comas.Activation_Cam_Auto := 1, [12].Comas.Distance_CPT_Presence_Produit := 520, [12].Comas.Consigne_Vitesse_Manu_Tour := 10.0, [12].Comas.Consigne_Acc_Decc_Manu_Tour := 10.0, [12].Comas.Mode_Decoreuse_Cam_Logique := 1, [12].Comas.Reserve_Real6 := 200.0, [13].Name := 'MIDOUX 44', [13].Comas.Pas_Machine := 60, [13].Comas.Came_Maitre[1].Master := 60.0, [13].Comas.Came_Maitre[1].Slave := 60.0, [13].Comas.Longueur_Came_Maitre := 2, [13].Comas.Tete.Stop_Cam_Logique_Degagement := 10.0, [13].Comas.Tete.Position_Degagement_H := 50.0, [13].Comas.Tete.Position_Degagement_V := 35.0, [13].Comas.Tete.Hauteur_Tete := -13, [13].Comas.Tete.Cam_Axe_Horizontal[1].Master := 1.0, [13].Comas.Tete.Cam_Axe_Horizontal[1].SegmentType := 1, [13].Comas.Tete.Cam_Axe_Horizontal[2].Master := 6.0, [13].Comas.Tete.Cam_Axe_Horizontal[2].Slave := 2.0, [13].Comas.Tete.Cam_Axe_Horizontal[3].Master := 21.0, [13].Comas.Tete.Cam_Axe_Horizontal[3].Slave := 27.0, [13].Comas.Tete.Cam_Axe_Horizontal[3].SegmentType := 1, [13].Comas.Tete.Cam_Axe_Horizontal[4].Master := 31.0,
        [13].Comas.Tete.Cam_Axe_Horizontal[4].Slave := 32.0, [13].Comas.Tete.Cam_Axe_Horizontal[5].Master := 36.0, [13].Comas.Tete.Cam_Axe_Horizontal[5].Slave := 32.0, [13].Comas.Tete.Cam_Axe_Horizontal[5].SegmentType := 1, [13].Comas.Tete.Cam_Axe_Horizontal[6].Master := 46.0, [13].Comas.Tete.Cam_Axe_Horizontal[6].Slave := 22.0, [13].Comas.Tete.Cam_Axe_Horizontal[6].SegmentType := 1, [13].Comas.Tete.Cam_Axe_Horizontal[7].Master := 60.0, [13].Comas.Tete.Cam_Axe_Vertical[1].Master := 1.0, [13].Comas.Tete.Cam_Axe_Vertical[2].Master := 6.0, [13].Comas.Tete.Cam_Axe_Vertical[3].Master := 11.0, [13].Comas.Tete.Cam_Axe_Vertical[3].SegmentType := 1, [13].Comas.Tete.Cam_Axe_Vertical[4].Master := 21.0, [13].Comas.Tete.Cam_Axe_Vertical[4].Slave := 3.0, [13].Comas.Tete.Cam_Axe_Vertical[5].Master := 41.0, [13].Comas.Tete.Cam_Axe_Vertical[5].Slave := 3.0, [13].Comas.Tete.Cam_Axe_Vertical[5].SegmentType := 1, [13].Comas.Tete.Cam_Axe_Vertical[6].Master := 56.0, [13].Comas.Tete.Cam_Axe_Vertical[7].Master := 60.0, [13].Comas.Tete.Longueur_Cam_Axe_H := 8, [13].Comas.Tete.Offset_Vertical_Gauche := 38.0, [13].Comas.Tete.Offset_Horizontal_Gauche := 95.0, [13].Comas.Tete.Cam_Axe_Horizontal_Pan.B.x := 1.0, [13].Comas.Tete.Cam_Axe_Horizontal_Pan.C.x := 5.0, [13].Comas.Tete.Cam_Axe_Horizontal_Pan.C.y := 2.0, [13].Comas.Tete.Cam_Axe_Horizontal_Pan.D.x := 15.0, [13].Comas.Tete.Cam_Axe_Horizontal_Pan.D.y := 25.0, [13].Comas.Tete.Cam_Axe_Horizontal_Pan.E.x := 10.0, [13].Comas.Tete.Cam_Axe_Horizontal_Pan.E.y := 5.0, [13].Comas.Tete.Cam_Axe_Horizontal_Pan.F.x := 5.0, [13].Comas.Tete.Cam_Axe_Horizontal_Pan.G.x := 10.0, [13].Comas.Tete.Cam_Axe_Horizontal_Pan.G.y := -10.0, [13].Comas.Tete.Cam_Axe_Vertical_Pan.K.x := -10.0, [13].Comas.Tete.Cam_Axe_Vertical_Pan.L.x := -10.0, [13].Comas.Tete.Cam_Axe_Vertical_Pan.L.y := 3.0, [13].Comas.Tete.Cam_Axe_Vertical_Pan.M.x := 5.0, [13].Comas.Tete.Cam_Axe_Vertical_Pan.M.y := 3.0, [13].Comas.Tete.Cam_Axe_Vertical_Pan.N.x := 10.0, [13].Comas.Tete.Offset_Vertical_Droit := 45.0, [13].Comas.Tete.Offset_Horizontal_Droit := 95.0, [13].Comas.Pompe.Start_Cam_Logique_Avance := -8.0, [13].Comas.Pompe.Stop_Cam_Logique_Avance := 7.0, [13].Comas.Pompe.Start_Cam_Logique_Recul := 7.0, [13].Comas.Pompe.Stop_Cam_Logique_Recul := 22.0, [13].Comas.Pompe.Consigne_Vitesse_Avance := 47.5, [13].Comas.Pompe.Consigne_Acc_Dec_Avance := 40.0, [13].Comas.Pompe.Consigne_Jerk_Avance := 100.0, [13].Comas.Pompe.Consigne_Vitesse_Recul := -28.0, [13].Comas.Pompe.Consigne_Acc_Dec_Recul := 40.0, [13].Comas.Pompe.Consigne_Jerk_Recul := 100.0, [13].Comas.Pompe.Points_Pan.O.x := -14.0, [13].Comas.Pompe.Points_Pan.Q.x := 15.0, [13].Comas.Pompe.Points_Pan.S.x := -4.0, [13].Comas.Pompe.Points_Pan.U.x := 15.0, [13].Comas.Pompe.Reserve_Bool1 := 1, [13].Comas.Rouleaux.Syncho_Pompe := 1, [13].Comas.Rouleaux.Consigne_Vitesse := 26.0, [13].Comas.Rouleaux.Consigne_Acc_Dec := 40.0, [13].Comas.Rouleaux.Consigne_Jerk := 100.0, [13].Comas.Rouleaux.Reserve_Real2 := 500.0,
        [13].Comas.Coupe_Fil.Start_Cam_Logique_Virtuelle := 11.0, [13].Comas.Coupe_Fil.Stop_Cam_Logique_Virtuelle := 21.0, [13].Comas.Coupe_Fil.Consigne_Vitesse_Virtuelle := 200.0, [13].Comas.Coupe_Fil.Consigne_Acc_Dec_Virtuelle := 1000.0, [13].Comas.Coupe_Fil.Consigne_Jerk_Virtuelle := 50.0, [13].Comas.Coupe_Fil.Cam_Axe[0].SegmentType := 1, [13].Comas.Coupe_Fil.Cam_Axe[1].Master := 180.0, [13].Comas.Coupe_Fil.Cam_Axe[1].Slave := 90.0, [13].Comas.Coupe_Fil.Cam_Axe[2].Master := 360.0, [13].Comas.Coupe_Fil.Cam_Axe[2].Slave := 360.0, [13].Comas.Coupe_Fil.Cam_Axe[2].SegmentType := 1, [13].Comas.Coupe_Fil.Points_Pan.W.x := 30.0, [13].Comas.Consigne_Vitesse_Manu_mm := 4.0, [13].Comas.Consigne_Acc_Decc_Manu_mm := 10.0, [13].Comas.Consigne_Jerk_Manu := 100.0, [13].Comas.Activation_Cam_Auto := 1, [13].Comas.Distance_CPT_Presence_Produit := 520, [13].Comas.Consigne_Vitesse_Manu_Tour := 10.0, [13].Comas.Consigne_Acc_Decc_Manu_Tour := 10.0, [13].Comas.Mode_Decoreuse_Cam_Logique := 1, [13].Comas.Reserve_Real3 := 1.0, [13].Comas.Reserve_Real4 := 1.0, [13].Comas.Reserve_Real5 := 5.0, [13].Comas.Reserve_Real6 := 200.0, [13].Reserve_Real2 := 200.0, [13].Reserve_Real3 := 10.0, [14].Name := 'MIDOUX 42', [14].Comas.Pas_Machine := 60, [14].Comas.Came_Maitre[1].Master := 60.0, [14].Comas.Came_Maitre[1].Slave := 60.0, [14].Comas.Longueur_Came_Maitre := 2, [14].Comas.Tete.Stop_Cam_Logique_Degagement := 10.0, [14].Comas.Tete.Position_Degagement_H := 50.0, [14].Comas.Tete.Position_Degagement_V := 35.0, [14].Comas.Tete.Hauteur_Tete := -1, [14].Comas.Tete.Cam_Axe_Horizontal[1].Master := 1.0, [14].Comas.Tete.Cam_Axe_Horizontal[1].SegmentType := 1, [14].Comas.Tete.Cam_Axe_Horizontal[2].Master := 6.0, [14].Comas.Tete.Cam_Axe_Horizontal[2].Slave := 2.0, [14].Comas.Tete.Cam_Axe_Horizontal[3].Master := 21.0, [14].Comas.Tete.Cam_Axe_Horizontal[3].Slave := 27.0, [14].Comas.Tete.Cam_Axe_Horizontal[3].SegmentType := 1, [14].Comas.Tete.Cam_Axe_Horizontal[4].Master := 31.0, [14].Comas.Tete.Cam_Axe_Horizontal[4].Slave := 32.0, [14].Comas.Tete.Cam_Axe_Horizontal[5].Master := 36.0, [14].Comas.Tete.Cam_Axe_Horizontal[5].Slave := 32.0, [14].Comas.Tete.Cam_Axe_Horizontal[5].SegmentType := 1, [14].Comas.Tete.Cam_Axe_Horizontal[6].Master := 46.0, [14].Comas.Tete.Cam_Axe_Horizontal[6].Slave := 22.0, [14].Comas.Tete.Cam_Axe_Horizontal[6].SegmentType := 1, [14].Comas.Tete.Cam_Axe_Horizontal[7].Master := 60.0, [14].Comas.Tete.Cam_Axe_Vertical[1].Master := 1.0, [14].Comas.Tete.Cam_Axe_Vertical[2].Master := 6.0, [14].Comas.Tete.Cam_Axe_Vertical[3].Master := 11.0, [14].Comas.Tete.Cam_Axe_Vertical[3].SegmentType := 1, [14].Comas.Tete.Cam_Axe_Vertical[4].Master := 21.0, [14].Comas.Tete.Cam_Axe_Vertical[4].Slave := 3.0, [14].Comas.Tete.Cam_Axe_Vertical[5].Master := 41.0, [14].Comas.Tete.Cam_Axe_Vertical[5].Slave := 3.0, [14].Comas.Tete.Cam_Axe_Vertical[5].SegmentType := 1,
        [14].Comas.Tete.Cam_Axe_Vertical[6].Master := 56.0, [14].Comas.Tete.Cam_Axe_Vertical[7].Master := 60.0, [14].Comas.Tete.Longueur_Cam_Axe_H := 8, [14].Comas.Tete.Offset_Vertical_Gauche := 38.0, [14].Comas.Tete.Offset_Horizontal_Gauche := 95.0, [14].Comas.Tete.Cam_Axe_Horizontal_Pan.B.x := 1.0, [14].Comas.Tete.Cam_Axe_Horizontal_Pan.C.x := 5.0, [14].Comas.Tete.Cam_Axe_Horizontal_Pan.C.y := 2.0, [14].Comas.Tete.Cam_Axe_Horizontal_Pan.D.x := 15.0, [14].Comas.Tete.Cam_Axe_Horizontal_Pan.D.y := 25.0, [14].Comas.Tete.Cam_Axe_Horizontal_Pan.E.x := 10.0, [14].Comas.Tete.Cam_Axe_Horizontal_Pan.E.y := 5.0, [14].Comas.Tete.Cam_Axe_Horizontal_Pan.F.x := 5.0, [14].Comas.Tete.Cam_Axe_Horizontal_Pan.G.x := 10.0, [14].Comas.Tete.Cam_Axe_Horizontal_Pan.G.y := -10.0, [14].Comas.Tete.Cam_Axe_Vertical_Pan.K.x := -10.0, [14].Comas.Tete.Cam_Axe_Vertical_Pan.L.x := -10.0, [14].Comas.Tete.Cam_Axe_Vertical_Pan.L.y := 3.0, [14].Comas.Tete.Cam_Axe_Vertical_Pan.M.x := 5.0, [14].Comas.Tete.Cam_Axe_Vertical_Pan.M.y := 3.0, [14].Comas.Tete.Cam_Axe_Vertical_Pan.N.x := 10.0, [14].Comas.Tete.Offset_Vertical_Droit := 45.0, [14].Comas.Tete.Offset_Horizontal_Droit := 95.0, [14].Comas.Pompe.Start_Cam_Logique_Avance := -8.0, [14].Comas.Pompe.Stop_Cam_Logique_Avance := 7.0, [14].Comas.Pompe.Start_Cam_Logique_Recul := 7.0, [14].Comas.Pompe.Stop_Cam_Logique_Recul := 22.0, [14].Comas.Pompe.Consigne_Vitesse_Avance := 42.6, [14].Comas.Pompe.Consigne_Acc_Dec_Avance := 40.0, [14].Comas.Pompe.Consigne_Jerk_Avance := 100.0, [14].Comas.Pompe.Consigne_Vitesse_Recul := -28.0, [14].Comas.Pompe.Consigne_Acc_Dec_Recul := 40.0, [14].Comas.Pompe.Consigne_Jerk_Recul := 100.0, [14].Comas.Pompe.Points_Pan.O.x := -14.0, [14].Comas.Pompe.Points_Pan.Q.x := 15.0, [14].Comas.Pompe.Points_Pan.S.x := -4.0, [14].Comas.Pompe.Points_Pan.U.x := 15.0, [14].Comas.Pompe.Reserve_Bool1 := 1, [14].Comas.Rouleaux.Consigne_Vitesse := 25.0, [14].Comas.Rouleaux.Consigne_Acc_Dec := 40.0, [14].Comas.Rouleaux.Consigne_Jerk := 100.0, [14].Comas.Rouleaux.Reserve_Real1 := -15.0, [14].Comas.Coupe_Fil.Start_Cam_Logique_Virtuelle := 11.0, [14].Comas.Coupe_Fil.Stop_Cam_Logique_Virtuelle := 21.0, [14].Comas.Coupe_Fil.Consigne_Vitesse_Virtuelle := 200.0, [14].Comas.Coupe_Fil.Consigne_Acc_Dec_Virtuelle := 1000.0, [14].Comas.Coupe_Fil.Consigne_Jerk_Virtuelle := 50.0, [14].Comas.Coupe_Fil.Cam_Axe[0].SegmentType := 1, [14].Comas.Coupe_Fil.Cam_Axe[1].Master := 180.0, [14].Comas.Coupe_Fil.Cam_Axe[1].Slave := 90.0, [14].Comas.Coupe_Fil.Cam_Axe[2].Master := 360.0, [14].Comas.Coupe_Fil.Cam_Axe[2].Slave := 360.0, [14].Comas.Coupe_Fil.Cam_Axe[2].SegmentType := 1, [14].Comas.Coupe_Fil.Points_Pan.W.x := 30.0, [14].Comas.Consigne_Vitesse_Manu_mm := 4.0, [14].Comas.Consigne_Acc_Decc_Manu_mm := 10.0, [14].Comas.Consigne_Jerk_Manu := 100.0, [14].Comas.Activation_Cam_Auto := 1, [14].Comas.Distance_CPT_Presence_Produit := 520, [14].Comas.Consigne_Vitesse_Manu_Tour := 10.0,
        [14].Comas.Consigne_Acc_Decc_Manu_Tour := 10.0, [14].Comas.Mode_Decoreuse_Cam_Logique := 1, [14].Comas.Reserve_Real6 := 200.0, [15].Name := 'COOKIE 311MIN010', [15].Comas.Pas_Machine := 95, [15].Comas.Came_Maitre[1].Master := 95.0, [15].Comas.Came_Maitre[1].Slave := 95.0, [15].Comas.Longueur_Came_Maitre := 2, [15].Comas.Tete.Stop_Cam_Logique_Degagement := 10.0, [15].Comas.Tete.Position_Degagement_H := 50.0, [15].Comas.Tete.Position_Degagement_V := 35.0, [15].Comas.Tete.Cam_Axe_Horizontal[1].Master := 1.0, [15].Comas.Tete.Cam_Axe_Horizontal[1].SegmentType := 1, [15].Comas.Tete.Cam_Axe_Horizontal[2].Master := 11.0, [15].Comas.Tete.Cam_Axe_Horizontal[2].Slave := 5.0, [15].Comas.Tete.Cam_Axe_Horizontal[3].Master := 41.0, [15].Comas.Tete.Cam_Axe_Horizontal[3].Slave := 35.0, [15].Comas.Tete.Cam_Axe_Horizontal[3].SegmentType := 1, [15].Comas.Tete.Cam_Axe_Horizontal[4].Master := 51.0, [15].Comas.Tete.Cam_Axe_Horizontal[4].Slave := 40.0, [15].Comas.Tete.Cam_Axe_Horizontal[5].Master := 61.0, [15].Comas.Tete.Cam_Axe_Horizontal[5].Slave := 40.0, [15].Comas.Tete.Cam_Axe_Horizontal[5].SegmentType := 1, [15].Comas.Tete.Cam_Axe_Horizontal[6].Master := 71.0, [15].Comas.Tete.Cam_Axe_Horizontal[6].Slave := 30.0, [15].Comas.Tete.Cam_Axe_Horizontal[6].SegmentType := 1, [15].Comas.Tete.Cam_Axe_Horizontal[7].Master := 95.0, [15].Comas.Tete.Cam_Axe_Vertical[1].Master := 1.0, [15].Comas.Tete.Cam_Axe_Vertical[2].Master := 11.0, [15].Comas.Tete.Cam_Axe_Vertical[3].Master := 41.0, [15].Comas.Tete.Cam_Axe_Vertical[3].SegmentType := 1, [15].Comas.Tete.Cam_Axe_Vertical[4].Master := 56.0, [15].Comas.Tete.Cam_Axe_Vertical[4].Slave := 10.0, [15].Comas.Tete.Cam_Axe_Vertical[5].Master := 66.0, [15].Comas.Tete.Cam_Axe_Vertical[5].Slave := 10.0, [15].Comas.Tete.Cam_Axe_Vertical[5].SegmentType := 1, [15].Comas.Tete.Cam_Axe_Vertical[6].Master := 86.0, [15].Comas.Tete.Cam_Axe_Vertical[7].Master := 95.0, [15].Comas.Tete.Longueur_Cam_Axe_H := 8, [15].Comas.Tete.Offset_Vertical_Gauche := 38.0, [15].Comas.Tete.Offset_Horizontal_Gauche := 95.0, [15].Comas.Tete.Cam_Axe_Horizontal_Pan.B.x := 1.0, [15].Comas.Tete.Cam_Axe_Horizontal_Pan.C.x := 10.0, [15].Comas.Tete.Cam_Axe_Horizontal_Pan.C.y := 5.0, [15].Comas.Tete.Cam_Axe_Horizontal_Pan.D.x := 30.0, [15].Comas.Tete.Cam_Axe_Horizontal_Pan.D.y := 30.0, [15].Comas.Tete.Cam_Axe_Horizontal_Pan.E.x := 10.0, [15].Comas.Tete.Cam_Axe_Horizontal_Pan.E.y := 5.0, [15].Comas.Tete.Cam_Axe_Horizontal_Pan.F.x := 10.0, [15].Comas.Tete.Cam_Axe_Horizontal_Pan.G.x := 10.0, [15].Comas.Tete.Cam_Axe_Horizontal_Pan.G.y := -10.0, [15].Comas.Tete.Cam_Axe_Vertical_Pan.L.x := 5.0, [15].Comas.Tete.Cam_Axe_Vertical_Pan.L.y := 10.0, [15].Comas.Tete.Cam_Axe_Vertical_Pan.M.x := 5.0, [15].Comas.Tete.Cam_Axe_Vertical_Pan.M.y := 10.0, [15].Comas.Tete.Cam_Axe_Vertical_Pan.N.x := 15.0, [15].Comas.Tete.Offset_Vertical_Droit := 45.0, [15].Comas.Tete.Offset_Horizontal_Droit := 95.0, [15].Comas.Pompe.Start_Cam_Logique_Avance := 1.0, [15].Comas.Pompe.Stop_Cam_Logique_Avance := 14.0,
        [15].Comas.Pompe.Start_Cam_Logique_Recul := 41.0, [15].Comas.Pompe.Stop_Cam_Logique_Recul := 41.0, [15].Comas.Pompe.Consigne_Vitesse_Avance := 13.9, [15].Comas.Pompe.Consigne_Acc_Dec_Avance := 40.0, [15].Comas.Pompe.Consigne_Jerk_Avance := 100.0, [15].Comas.Pompe.Consigne_Acc_Dec_Recul := 40.0, [15].Comas.Pompe.Consigne_Jerk_Recul := 100.0, [15].Comas.Pompe.Points_Pan.O.x := -10.0, [15].Comas.Pompe.Points_Pan.Q.x := 13.0, [15].Comas.Pompe.Reserve_Bool1 := 1, [15].Comas.Rouleaux.Syncho_Pompe := 1, [15].Comas.Rouleaux.Consigne_Vitesse := 31.0, [15].Comas.Rouleaux.Consigne_Acc_Dec := 40.0, [15].Comas.Rouleaux.Consigne_Jerk := 100.0, [15].Comas.Rouleaux.Reserve_Real1 := -15.0, [15].Comas.Coupe_Fil.Activation := 1, [15].Comas.Coupe_Fil.Start_Cam_Logique_Virtuelle := 11.0, [15].Comas.Coupe_Fil.Stop_Cam_Logique_Virtuelle := 21.0, [15].Comas.Coupe_Fil.Consigne_Vitesse_Virtuelle := 250.0, [15].Comas.Coupe_Fil.Consigne_Acc_Dec_Virtuelle := 1000.0, [15].Comas.Coupe_Fil.Consigne_Jerk_Virtuelle := 50.0, [15].Comas.Coupe_Fil.Cam_Axe[0].SegmentType := 1, [15].Comas.Coupe_Fil.Cam_Axe[1].Master := 180.0, [15].Comas.Coupe_Fil.Cam_Axe[1].Slave := 180.0, [15].Comas.Coupe_Fil.Cam_Axe[2].Master := 250.0, [15].Comas.Coupe_Fil.Cam_Axe[2].Slave := 180.0, [15].Comas.Coupe_Fil.Cam_Axe[2].SegmentType := 1, [15].Comas.Coupe_Fil.Cam_Axe[3].Master := 360.0, [15].Comas.Coupe_Fil.Cam_Axe[3].Slave := 360.0, [15].Comas.Coupe_Fil.Cam_Axe[3].SegmentType := 1, [15].Comas.Coupe_Fil.Cam_Axe[4].SegmentType := 1, [15].Comas.Coupe_Fil.Points_Pan.W.x := -40.0, [15].Comas.Coupe_Fil.Reserve_Bool1 := 1, [15].Comas.Consigne_Vitesse_Manu_mm := 2.0, [15].Comas.Consigne_Acc_Decc_Manu_mm := 10.0, [15].Comas.Consigne_Jerk_Manu := 100.0, [15].Comas.Activation_Cam_Auto := 1, [15].Comas.Distance_CPT_Presence_Produit := 520, [15].Comas.Consigne_Vitesse_Manu_Tour := 10.0, [15].Comas.Consigne_Acc_Decc_Manu_Tour := 10.0, [15].Comas.Mode_Decoreuse_Cam_Logique := 1, [15].Comas.Reserve_Real6 := 200.0, [16].Name := 'PALET CAJOU 318PJL002', [16].Comas.Pas_Machine := 70, [16].Comas.Came_Maitre[1].Master := 70.0, [16].Comas.Came_Maitre[1].Slave := 70.0, [16].Comas.Longueur_Came_Maitre := 2, [16].Comas.Tete.Stop_Cam_Logique_Degagement := 10.0, [16].Comas.Tete.Position_Degagement_H := 50.0, [16].Comas.Tete.Position_Degagement_V := 35.0, [16].Comas.Tete.Hauteur_Tete := -2, [16].Comas.Tete.Cam_Axe_Horizontal[1].Master := 1.0, [16].Comas.Tete.Cam_Axe_Horizontal[1].SegmentType := 1, [16].Comas.Tete.Cam_Axe_Horizontal[2].Master := 6.0, [16].Comas.Tete.Cam_Axe_Horizontal[2].Slave := 2.0, [16].Comas.Tete.Cam_Axe_Horizontal[3].Master := 21.0, [16].Comas.Tete.Cam_Axe_Horizontal[3].Slave := 27.0, [16].Comas.Tete.Cam_Axe_Horizontal[3].SegmentType := 1, [16].Comas.Tete.Cam_Axe_Horizontal[4].Master := 31.0, [16].Comas.Tete.Cam_Axe_Horizontal[4].Slave := 32.0,
        [16].Comas.Tete.Cam_Axe_Horizontal[5].Master := 36.0, [16].Comas.Tete.Cam_Axe_Horizontal[5].Slave := 32.0, [16].Comas.Tete.Cam_Axe_Horizontal[5].SegmentType := 1, [16].Comas.Tete.Cam_Axe_Horizontal[6].Master := 46.0, [16].Comas.Tete.Cam_Axe_Horizontal[6].Slave := 22.0, [16].Comas.Tete.Cam_Axe_Horizontal[6].SegmentType := 1, [16].Comas.Tete.Cam_Axe_Horizontal[7].Master := 70.0, [16].Comas.Tete.Cam_Axe_Vertical[1].Master := 1.0, [16].Comas.Tete.Cam_Axe_Vertical[2].Master := 6.0, [16].Comas.Tete.Cam_Axe_Vertical[3].Master := 11.0, [16].Comas.Tete.Cam_Axe_Vertical[3].SegmentType := 1, [16].Comas.Tete.Cam_Axe_Vertical[4].Master := 21.0, [16].Comas.Tete.Cam_Axe_Vertical[4].Slave := 5.0, [16].Comas.Tete.Cam_Axe_Vertical[5].Master := 41.0, [16].Comas.Tete.Cam_Axe_Vertical[5].Slave := 5.0, [16].Comas.Tete.Cam_Axe_Vertical[5].SegmentType := 1, [16].Comas.Tete.Cam_Axe_Vertical[6].Master := 56.0, [16].Comas.Tete.Cam_Axe_Vertical[7].Master := 70.0, [16].Comas.Tete.Longueur_Cam_Axe_H := 8, [16].Comas.Tete.Offset_Vertical_Gauche := 38.0, [16].Comas.Tete.Offset_Horizontal_Gauche := 95.0, [16].Comas.Tete.Cam_Axe_Horizontal_Pan.B.x := 1.0, [16].Comas.Tete.Cam_Axe_Horizontal_Pan.C.x := 5.0, [16].Comas.Tete.Cam_Axe_Horizontal_Pan.C.y := 2.0, [16].Comas.Tete.Cam_Axe_Horizontal_Pan.D.x := 15.0, [16].Comas.Tete.Cam_Axe_Horizontal_Pan.D.y := 25.0, [16].Comas.Tete.Cam_Axe_Horizontal_Pan.E.x := 10.0, [16].Comas.Tete.Cam_Axe_Horizontal_Pan.E.y := 5.0, [16].Comas.Tete.Cam_Axe_Horizontal_Pan.F.x := 5.0, [16].Comas.Tete.Cam_Axe_Horizontal_Pan.G.x := 10.0, [16].Comas.Tete.Cam_Axe_Horizontal_Pan.G.y := -10.0, [16].Comas.Tete.Cam_Axe_Vertical_Pan.K.x := -10.0, [16].Comas.Tete.Cam_Axe_Vertical_Pan.L.x := -10.0, [16].Comas.Tete.Cam_Axe_Vertical_Pan.L.y := 5.0, [16].Comas.Tete.Cam_Axe_Vertical_Pan.M.x := 5.0, [16].Comas.Tete.Cam_Axe_Vertical_Pan.M.y := 5.0, [16].Comas.Tete.Cam_Axe_Vertical_Pan.N.x := 10.0, [16].Comas.Tete.Offset_Vertical_Droit := 45.0, [16].Comas.Tete.Offset_Horizontal_Droit := 95.0, [16].Comas.Pompe.Start_Cam_Logique_Avance := -6.0, [16].Comas.Pompe.Stop_Cam_Logique_Avance := 12.0, [16].Comas.Pompe.Start_Cam_Logique_Recul := 19.0, [16].Comas.Pompe.Stop_Cam_Logique_Recul := 49.0, [16].Comas.Pompe.Consigne_Vitesse_Avance := 41.5, [16].Comas.Pompe.Consigne_Acc_Dec_Avance := 40.0, [16].Comas.Pompe.Consigne_Jerk_Avance := 100.0, [16].Comas.Pompe.Consigne_Vitesse_Recul := -14.0, [16].Comas.Pompe.Consigne_Acc_Dec_Recul := 40.0, [16].Comas.Pompe.Consigne_Jerk_Recul := 100.0, [16].Comas.Pompe.Points_Pan.O.x := -12.0, [16].Comas.Pompe.Points_Pan.Q.x := 18.0, [16].Comas.Pompe.Points_Pan.S.x := 8.0, [16].Comas.Pompe.Points_Pan.U.x := 30.0, [16].Comas.Pompe.Reserve_Bool1 := 1, [16].Comas.Rouleaux.Syncho_Pompe := 1, [16].Comas.Rouleaux.Consigne_Vitesse := 25.0, [16].Comas.Rouleaux.Consigne_Acc_Dec := 40.0, [16].Comas.Rouleaux.Consigne_Jerk := 100.0, [16].Comas.Rouleaux.Reserve_Real1 := -15.0, [16].Comas.Coupe_Fil.Start_Cam_Logique_Virtuelle := 11.0,
        [16].Comas.Coupe_Fil.Stop_Cam_Logique_Virtuelle := 21.0, [16].Comas.Coupe_Fil.Consigne_Vitesse_Virtuelle := 200.0, [16].Comas.Coupe_Fil.Consigne_Acc_Dec_Virtuelle := 1000.0, [16].Comas.Coupe_Fil.Consigne_Jerk_Virtuelle := 50.0, [16].Comas.Coupe_Fil.Cam_Axe[0].SegmentType := 1, [16].Comas.Coupe_Fil.Cam_Axe[1].Master := 180.0, [16].Comas.Coupe_Fil.Cam_Axe[1].Slave := 90.0, [16].Comas.Coupe_Fil.Cam_Axe[2].Master := 360.0, [16].Comas.Coupe_Fil.Cam_Axe[2].Slave := 360.0, [16].Comas.Coupe_Fil.Cam_Axe[2].SegmentType := 1, [16].Comas.Coupe_Fil.Points_Pan.W.x := 30.0, [16].Comas.Consigne_Vitesse_Manu_mm := 4.0, [16].Comas.Consigne_Acc_Decc_Manu_mm := 10.0, [16].Comas.Consigne_Jerk_Manu := 100.0, [16].Comas.Activation_Cam_Auto := 1, [16].Comas.Distance_CPT_Presence_Produit := 520, [16].Comas.Consigne_Vitesse_Manu_Tour := 10.0, [16].Comas.Consigne_Acc_Decc_Manu_Tour := 10.0, [16].Comas.Mode_Decoreuse_Cam_Logique := 1, [16].Comas.Reserve_Real6 := 200.0, [17].Name := 'PASSION 311PAS004', [17].Comas.Pas_Machine := 85, [17].Comas.Came_Maitre[1].Master := 85.0, [17].Comas.Came_Maitre[1].Slave := 85.0, [17].Comas.Longueur_Came_Maitre := 2, [17].Comas.Tete.Stop_Cam_Logique_Degagement := 10.0, [17].Comas.Tete.Position_Degagement_H := 50.0, [17].Comas.Tete.Position_Degagement_V := 35.0, [17].Comas.Tete.Hauteur_Tete := -4, [17].Comas.Tete.Cam_Axe_Horizontal[1].Master := 1.0, [17].Comas.Tete.Cam_Axe_Horizontal[1].SegmentType := 1, [17].Comas.Tete.Cam_Axe_Horizontal[2].Master := 6.0, [17].Comas.Tete.Cam_Axe_Horizontal[2].Slave := 5.0, [17].Comas.Tete.Cam_Axe_Horizontal[3].Master := 36.0, [17].Comas.Tete.Cam_Axe_Horizontal[3].Slave := 75.0, [17].Comas.Tete.Cam_Axe_Horizontal[3].SegmentType := 1, [17].Comas.Tete.Cam_Axe_Horizontal[4].Master := 46.0, [17].Comas.Tete.Cam_Axe_Horizontal[4].Slave := 85.0, [17].Comas.Tete.Cam_Axe_Horizontal[5].Master := 51.0, [17].Comas.Tete.Cam_Axe_Horizontal[5].Slave := 85.0, [17].Comas.Tete.Cam_Axe_Horizontal[5].SegmentType := 1, [17].Comas.Tete.Cam_Axe_Horizontal[6].Master := 61.0, [17].Comas.Tete.Cam_Axe_Horizontal[6].Slave := 75.0, [17].Comas.Tete.Cam_Axe_Horizontal[6].SegmentType := 1, [17].Comas.Tete.Cam_Axe_Horizontal[7].Master := 85.0, [17].Comas.Tete.Cam_Axe_Vertical[0].Slave := 15.0, [17].Comas.Tete.Cam_Axe_Vertical[1].Master := 1.0, [17].Comas.Tete.Cam_Axe_Vertical[1].Slave := 15.0, [17].Comas.Tete.Cam_Axe_Vertical[2].Master := 6.0, [17].Comas.Tete.Cam_Axe_Vertical[2].Slave := 15.0, [17].Comas.Tete.Cam_Axe_Vertical[3].Master := 46.0, [17].Comas.Tete.Cam_Axe_Vertical[3].Slave := 15.0, [17].Comas.Tete.Cam_Axe_Vertical[3].SegmentType := 1, [17].Comas.Tete.Cam_Axe_Vertical[4].Master := 56.0, [17].Comas.Tete.Cam_Axe_Vertical[4].Slave := 20.0, [17].Comas.Tete.Cam_Axe_Vertical[5].Master := 66.0, [17].Comas.Tete.Cam_Axe_Vertical[5].Slave := 20.0, [17].Comas.Tete.Cam_Axe_Vertical[5].SegmentType := 1, [17].Comas.Tete.Cam_Axe_Vertical[6].Master := 81.0, [17].Comas.Tete.Cam_Axe_Vertical[6].Slave := 15.0,
        [17].Comas.Tete.Cam_Axe_Vertical[7].Master := 85.0, [17].Comas.Tete.Cam_Axe_Vertical[7].Slave := 15.0, [17].Comas.Tete.Longueur_Cam_Axe_H := 8, [17].Comas.Tete.Offset_Vertical_Gauche := 38.0, [17].Comas.Tete.Offset_Horizontal_Gauche := 95.0, [17].Comas.Tete.Cam_Axe_Horizontal_Pan.B.x := 1.0, [17].Comas.Tete.Cam_Axe_Horizontal_Pan.C.x := 5.0, [17].Comas.Tete.Cam_Axe_Horizontal_Pan.C.y := 5.0, [17].Comas.Tete.Cam_Axe_Horizontal_Pan.D.x := 30.0, [17].Comas.Tete.Cam_Axe_Horizontal_Pan.D.y := 70.0, [17].Comas.Tete.Cam_Axe_Horizontal_Pan.E.x := 10.0, [17].Comas.Tete.Cam_Axe_Horizontal_Pan.E.y := 10.0, [17].Comas.Tete.Cam_Axe_Horizontal_Pan.F.x := 5.0, [17].Comas.Tete.Cam_Axe_Horizontal_Pan.G.x := 10.0, [17].Comas.Tete.Cam_Axe_Horizontal_Pan.G.y := -10.0, [17].Comas.Tete.Cam_Axe_Vertical_Pan.H.y := 15.0, [17].Comas.Tete.Cam_Axe_Vertical_Pan.I.y := 15.0, [17].Comas.Tete.Cam_Axe_Vertical_Pan.J.y := 15.0, [17].Comas.Tete.Cam_Axe_Vertical_Pan.K.x := 10.0, [17].Comas.Tete.Cam_Axe_Vertical_Pan.K.y := 15.0, [17].Comas.Tete.Cam_Axe_Vertical_Pan.L.x := 10.0, [17].Comas.Tete.Cam_Axe_Vertical_Pan.L.y := 20.0, [17].Comas.Tete.Cam_Axe_Vertical_Pan.M.x := 15.0, [17].Comas.Tete.Cam_Axe_Vertical_Pan.M.y := 20.0, [17].Comas.Tete.Cam_Axe_Vertical_Pan.N.x := 20.0, [17].Comas.Tete.Cam_Axe_Vertical_Pan.N.y := 15.0, [17].Comas.Tete.Offset_Vertical_Droit := 45.0, [17].Comas.Tete.Offset_Horizontal_Droit := 95.0, [17].Comas.Pompe.Start_Cam_Logique_Avance := -15.5, [17].Comas.Pompe.Stop_Cam_Logique_Avance := 29.5, [17].Comas.Pompe.Start_Cam_Logique_Recul := 30.0, [17].Comas.Pompe.Stop_Cam_Logique_Recul := 50.0, [17].Comas.Pompe.Consigne_Vitesse_Avance := 5.0, [17].Comas.Pompe.Consigne_Acc_Dec_Avance := 40.0, [17].Comas.Pompe.Consigne_Jerk_Avance := 100.0, [17].Comas.Pompe.Consigne_Vitesse_Recul := -4.0, [17].Comas.Pompe.Consigne_Acc_Dec_Recul := 40.0, [17].Comas.Pompe.Consigne_Jerk_Recul := 100.0, [17].Comas.Pompe.Points_Pan.O.x := -21.5, [17].Comas.Pompe.Points_Pan.Q.x := 45.0, [17].Comas.Pompe.Points_Pan.S.x := -16.0, [17].Comas.Pompe.Points_Pan.U.x := 20.0, [17].Comas.Pompe.Reserve_Bool1 := 1, [17].Comas.Rouleaux.Syncho_Pompe := 1, [17].Comas.Rouleaux.Consigne_Vitesse := 25.0, [17].Comas.Rouleaux.Consigne_Acc_Dec := 40.0, [17].Comas.Rouleaux.Consigne_Jerk := 100.0, [17].Comas.Coupe_Fil.Start_Cam_Logique_Virtuelle := 11.0, [17].Comas.Coupe_Fil.Stop_Cam_Logique_Virtuelle := 21.0, [17].Comas.Coupe_Fil.Consigne_Vitesse_Virtuelle := 200.0, [17].Comas.Coupe_Fil.Consigne_Acc_Dec_Virtuelle := 1000.0, [17].Comas.Coupe_Fil.Consigne_Jerk_Virtuelle := 50.0, [17].Comas.Coupe_Fil.Cam_Axe[0].SegmentType := 1, [17].Comas.Coupe_Fil.Cam_Axe[1].Master := 180.0, [17].Comas.Coupe_Fil.Cam_Axe[1].Slave := 90.0, [17].Comas.Coupe_Fil.Cam_Axe[2].Master := 360.0, [17].Comas.Coupe_Fil.Cam_Axe[2].Slave := 360.0, [17].Comas.Coupe_Fil.Cam_Axe[2].SegmentType := 1, [17].Comas.Coupe_Fil.Points_Pan.W.x := 30.0, [17].Comas.Consigne_Vitesse_Manu_mm := 4.0,
        [17].Comas.Consigne_Acc_Decc_Manu_mm := 10.0, [17].Comas.Consigne_Jerk_Manu := 100.0, [17].Comas.Activation_Cam_Auto := 1, [17].Comas.Distance_CPT_Presence_Produit := 520, [17].Comas.Consigne_Vitesse_Manu_Tour := 10.0, [17].Comas.Consigne_Acc_Decc_Manu_Tour := 10.0, [17].Comas.Mode_Decoreuse_Cam_Logique := 1, [17].Comas.Reserve_Real6 := 200.0, [18].Name := '314PJL010 LANGUE 40', [18].Comas.Pas_Machine := 67, [18].Comas.Came_Maitre[1].Master := 67.0, [18].Comas.Came_Maitre[1].Slave := 67.0, [18].Comas.Longueur_Came_Maitre := 2, [18].Comas.Tete.Stop_Cam_Logique_Degagement := 10.0, [18].Comas.Tete.Position_Degagement_H := 50.0, [18].Comas.Tete.Position_Degagement_V := 35.0, [18].Comas.Tete.Hauteur_Tete := -3, [18].Comas.Tete.Cam_Axe_Horizontal[1].Master := 1.0, [18].Comas.Tete.Cam_Axe_Horizontal[1].SegmentType := 1, [18].Comas.Tete.Cam_Axe_Horizontal[2].Master := 6.0, [18].Comas.Tete.Cam_Axe_Horizontal[2].Slave := 2.0, [18].Comas.Tete.Cam_Axe_Horizontal[3].Master := 31.0, [18].Comas.Tete.Cam_Axe_Horizontal[3].Slave := 27.0, [18].Comas.Tete.Cam_Axe_Horizontal[3].SegmentType := 1, [18].Comas.Tete.Cam_Axe_Horizontal[4].Master := 41.0, [18].Comas.Tete.Cam_Axe_Horizontal[4].Slave := 37.0, [18].Comas.Tete.Cam_Axe_Horizontal[5].Master := 46.0, [18].Comas.Tete.Cam_Axe_Horizontal[5].Slave := 37.0, [18].Comas.Tete.Cam_Axe_Horizontal[5].SegmentType := 1, [18].Comas.Tete.Cam_Axe_Horizontal[6].Master := 56.0, [18].Comas.Tete.Cam_Axe_Horizontal[6].Slave := 27.0, [18].Comas.Tete.Cam_Axe_Horizontal[6].SegmentType := 1, [18].Comas.Tete.Cam_Axe_Horizontal[7].Master := 67.0, [18].Comas.Tete.Cam_Axe_Vertical[1].Master := 1.0, [18].Comas.Tete.Cam_Axe_Vertical[2].Master := 6.0, [18].Comas.Tete.Cam_Axe_Vertical[3].Master := 21.0, [18].Comas.Tete.Cam_Axe_Vertical[3].SegmentType := 1, [18].Comas.Tete.Cam_Axe_Vertical[4].Master := 31.0, [18].Comas.Tete.Cam_Axe_Vertical[4].Slave := 1.0, [18].Comas.Tete.Cam_Axe_Vertical[5].Master := 51.0, [18].Comas.Tete.Cam_Axe_Vertical[5].Slave := 10.0, [18].Comas.Tete.Cam_Axe_Vertical[5].SegmentType := 1, [18].Comas.Tete.Cam_Axe_Vertical[6].Master := 66.0, [18].Comas.Tete.Cam_Axe_Vertical[7].Master := 67.0, [18].Comas.Tete.Longueur_Cam_Axe_H := 8, [18].Comas.Tete.Offset_Vertical_Gauche := 38.0, [18].Comas.Tete.Offset_Horizontal_Gauche := 95.0, [18].Comas.Tete.Cam_Axe_Horizontal_Pan.B.x := 1.0, [18].Comas.Tete.Cam_Axe_Horizontal_Pan.C.x := 5.0, [18].Comas.Tete.Cam_Axe_Horizontal_Pan.C.y := 2.0, [18].Comas.Tete.Cam_Axe_Horizontal_Pan.D.x := 25.0, [18].Comas.Tete.Cam_Axe_Horizontal_Pan.D.y := 25.0, [18].Comas.Tete.Cam_Axe_Horizontal_Pan.E.x := 10.0, [18].Comas.Tete.Cam_Axe_Horizontal_Pan.E.y := 10.0, [18].Comas.Tete.Cam_Axe_Horizontal_Pan.F.x := 5.0, [18].Comas.Tete.Cam_Axe_Horizontal_Pan.G.x := 10.0, [18].Comas.Tete.Cam_Axe_Horizontal_Pan.G.y := -10.0, [18].Comas.Tete.Cam_Axe_Vertical_Pan.K.x := -10.0, [18].Comas.Tete.Cam_Axe_Vertical_Pan.L.x := -10.0, [18].Comas.Tete.Cam_Axe_Vertical_Pan.L.y := 1.0,
        [18].Comas.Tete.Cam_Axe_Vertical_Pan.M.x := 5.0, [18].Comas.Tete.Cam_Axe_Vertical_Pan.M.y := 10.0, [18].Comas.Tete.Cam_Axe_Vertical_Pan.N.x := 10.0, [18].Comas.Tete.Offset_Vertical_Droit := 45.0, [18].Comas.Tete.Offset_Horizontal_Droit := 95.0, [18].Comas.Pompe.Start_Cam_Logique_Avance := -9.0, [18].Comas.Pompe.Stop_Cam_Logique_Avance := 16.0, [18].Comas.Pompe.Start_Cam_Logique_Recul := 21.0, [18].Comas.Pompe.Stop_Cam_Logique_Recul := 33.0, [18].Comas.Pompe.Consigne_Vitesse_Avance := 15.6, [18].Comas.Pompe.Consigne_Acc_Dec_Avance := 40.0, [18].Comas.Pompe.Consigne_Jerk_Avance := 100.0, [18].Comas.Pompe.Consigne_Vitesse_Recul := -18.0, [18].Comas.Pompe.Consigne_Acc_Dec_Recul := 40.0, [18].Comas.Pompe.Consigne_Jerk_Recul := 100.0, [18].Comas.Pompe.Points_Pan.O.x := -15.0, [18].Comas.Pompe.Points_Pan.Q.x := 25.0, [18].Comas.Pompe.Points_Pan.U.x := 12.0, [18].Comas.Pompe.Reserve_Bool1 := 1, [18].Comas.Rouleaux.Syncho_Pompe := 1, [18].Comas.Rouleaux.Consigne_Vitesse := 25.0, [18].Comas.Rouleaux.Consigne_Acc_Dec := 40.0, [18].Comas.Rouleaux.Consigne_Jerk := 100.0, [18].Comas.Coupe_Fil.Start_Cam_Logique_Virtuelle := 11.0, [18].Comas.Coupe_Fil.Stop_Cam_Logique_Virtuelle := 21.0, [18].Comas.Coupe_Fil.Consigne_Vitesse_Virtuelle := 200.0, [18].Comas.Coupe_Fil.Consigne_Acc_Dec_Virtuelle := 1000.0, [18].Comas.Coupe_Fil.Consigne_Jerk_Virtuelle := 50.0, [18].Comas.Coupe_Fil.Cam_Axe[0].SegmentType := 1, [18].Comas.Coupe_Fil.Cam_Axe[1].Master := 180.0, [18].Comas.Coupe_Fil.Cam_Axe[1].Slave := 90.0, [18].Comas.Coupe_Fil.Cam_Axe[2].Master := 360.0, [18].Comas.Coupe_Fil.Cam_Axe[2].Slave := 360.0, [18].Comas.Coupe_Fil.Cam_Axe[2].SegmentType := 1, [18].Comas.Coupe_Fil.Points_Pan.W.x := 30.0, [18].Comas.Consigne_Vitesse_Manu_mm := 4.0, [18].Comas.Consigne_Acc_Decc_Manu_mm := 10.0, [18].Comas.Consigne_Jerk_Manu := 100.0, [18].Comas.Activation_Cam_Auto := 1, [18].Comas.Distance_CPT_Presence_Produit := 520, [18].Comas.Consigne_Vitesse_Manu_Tour := 10.0, [18].Comas.Consigne_Acc_Decc_Manu_Tour := 10.0, [18].Comas.Mode_Decoreuse_Cam_Logique := 1, [18].Comas.Reserve_Real6 := 200.0, [19].Name := 'MERING ETOIL ', [19].Comas.Pas_Machine := 54, [19].Comas.Came_Maitre[1].Master := 54.0, [19].Comas.Came_Maitre[1].Slave := 54.0, [19].Comas.Longueur_Came_Maitre := 2, [19].Comas.Tete.Stop_Cam_Logique_Degagement := 10.0, [19].Comas.Tete.Position_Degagement_H := 50.0, [19].Comas.Tete.Position_Degagement_V := 35.0, [19].Comas.Tete.Hauteur_Tete := -2, [19].Comas.Tete.Cam_Axe_Horizontal[1].Master := 1.0, [19].Comas.Tete.Cam_Axe_Horizontal[1].SegmentType := 1, [19].Comas.Tete.Cam_Axe_Horizontal[2].Master := 6.0, [19].Comas.Tete.Cam_Axe_Horizontal[2].Slave := 2.0, [19].Comas.Tete.Cam_Axe_Horizontal[3].Master := 21.0, [19].Comas.Tete.Cam_Axe_Horizontal[3].Slave := 20.0, [19].Comas.Tete.Cam_Axe_Horizontal[3].SegmentType := 1,
        [19].Comas.Tete.Cam_Axe_Horizontal[4].Master := 26.0, [19].Comas.Tete.Cam_Axe_Horizontal[4].Slave := 25.0, [19].Comas.Tete.Cam_Axe_Horizontal[5].Master := 34.0, [19].Comas.Tete.Cam_Axe_Horizontal[5].Slave := 25.0, [19].Comas.Tete.Cam_Axe_Horizontal[5].SegmentType := 1, [19].Comas.Tete.Cam_Axe_Horizontal[6].Master := 44.0, [19].Comas.Tete.Cam_Axe_Horizontal[6].Slave := 20.0, [19].Comas.Tete.Cam_Axe_Horizontal[6].SegmentType := 1, [19].Comas.Tete.Cam_Axe_Horizontal[7].Master := 54.0, [19].Comas.Tete.Cam_Axe_Vertical[1].Master := 1.0, [19].Comas.Tete.Cam_Axe_Vertical[2].Master := 6.0, [19].Comas.Tete.Cam_Axe_Vertical[3].Master := 21.0, [19].Comas.Tete.Cam_Axe_Vertical[3].SegmentType := 1, [19].Comas.Tete.Cam_Axe_Vertical[4].Master := 31.0, [19].Comas.Tete.Cam_Axe_Vertical[4].Slave := 8.0, [19].Comas.Tete.Cam_Axe_Vertical[5].Master := 39.0, [19].Comas.Tete.Cam_Axe_Vertical[5].Slave := 8.0, [19].Comas.Tete.Cam_Axe_Vertical[5].SegmentType := 1, [19].Comas.Tete.Cam_Axe_Vertical[6].Master := 52.0, [19].Comas.Tete.Cam_Axe_Vertical[7].Master := 54.0, [19].Comas.Tete.Longueur_Cam_Axe_H := 8, [19].Comas.Tete.Offset_Vertical_Gauche := 38.0, [19].Comas.Tete.Offset_Horizontal_Gauche := 95.0, [19].Comas.Tete.Cam_Axe_Horizontal_Pan.B.x := 1.0, [19].Comas.Tete.Cam_Axe_Horizontal_Pan.C.x := 5.0, [19].Comas.Tete.Cam_Axe_Horizontal_Pan.C.y := 2.0, [19].Comas.Tete.Cam_Axe_Horizontal_Pan.D.x := 15.0, [19].Comas.Tete.Cam_Axe_Horizontal_Pan.D.y := 15.0, [19].Comas.Tete.Cam_Axe_Horizontal_Pan.E.x := 5.0, [19].Comas.Tete.Cam_Axe_Horizontal_Pan.E.y := 5.0, [19].Comas.Tete.Cam_Axe_Horizontal_Pan.F.x := 8.0, [19].Comas.Tete.Cam_Axe_Horizontal_Pan.G.x := 10.0, [19].Comas.Tete.Cam_Axe_Horizontal_Pan.G.y := -5.0, [19].Comas.Tete.Cam_Axe_Vertical_Pan.L.x := 5.0, [19].Comas.Tete.Cam_Axe_Vertical_Pan.L.y := 8.0, [19].Comas.Tete.Cam_Axe_Vertical_Pan.M.x := 5.0, [19].Comas.Tete.Cam_Axe_Vertical_Pan.M.y := 8.0, [19].Comas.Tete.Cam_Axe_Vertical_Pan.N.x := 8.0, [19].Comas.Tete.Offset_Vertical_Droit := 45.0, [19].Comas.Tete.Offset_Horizontal_Droit := 95.0, [19].Comas.Tete.Reserve_Real1 := 3.0, [19].Comas.Pompe.Start_Cam_Logique_Avance := -14.0, [19].Comas.Pompe.Stop_Cam_Logique_Avance := 16.0, [19].Comas.Pompe.Start_Cam_Logique_Recul := 16.0, [19].Comas.Pompe.Stop_Cam_Logique_Recul := 36.0, [19].Comas.Pompe.Consigne_Vitesse_Avance := 20.6, [19].Comas.Pompe.Consigne_Acc_Dec_Avance := 40.0, [19].Comas.Pompe.Consigne_Jerk_Avance := 100.0, [19].Comas.Pompe.Consigne_Vitesse_Recul := -20.5, [19].Comas.Pompe.Consigne_Acc_Dec_Recul := 40.0, [19].Comas.Pompe.Consigne_Jerk_Recul := 100.0, [19].Comas.Pompe.Points_Pan.O.x := -20.0, [19].Comas.Pompe.Points_Pan.Q.x := 30.0, [19].Comas.Pompe.Points_Pan.S.x := -5.0, [19].Comas.Pompe.Points_Pan.U.x := 20.0, [19].Comas.Pompe.Reserve_Bool1 := 1, [19].Comas.Rouleaux.Syncho_Pompe := 1, [19].Comas.Rouleaux.Consigne_Vitesse := 30.0, [19].Comas.Rouleaux.Consigne_Acc_Dec := 40.0, [19].Comas.Rouleaux.Consigne_Jerk := 100.0,
        [19].Comas.Coupe_Fil.Start_Cam_Logique_Virtuelle := 16.0, [19].Comas.Coupe_Fil.Stop_Cam_Logique_Virtuelle := 26.0, [19].Comas.Coupe_Fil.Consigne_Vitesse_Virtuelle := 200.0, [19].Comas.Coupe_Fil.Consigne_Acc_Dec_Virtuelle := 1000.0, [19].Comas.Coupe_Fil.Consigne_Jerk_Virtuelle := 50.0, [19].Comas.Coupe_Fil.Cam_Axe[0].SegmentType := 1, [19].Comas.Coupe_Fil.Cam_Axe[1].Master := 180.0, [19].Comas.Coupe_Fil.Cam_Axe[1].Slave := 90.0, [19].Comas.Coupe_Fil.Cam_Axe[2].Master := 360.0, [19].Comas.Coupe_Fil.Cam_Axe[2].Slave := 360.0, [19].Comas.Coupe_Fil.Cam_Axe[2].SegmentType := 1, [19].Comas.Coupe_Fil.Points_Pan.W.x := 30.0, [19].Comas.Consigne_Vitesse_Manu_mm := 2.0, [19].Comas.Consigne_Acc_Decc_Manu_mm := 10.0, [19].Comas.Consigne_Jerk_Manu := 100.0, [19].Comas.Activation_Cam_Auto := 1, [19].Comas.Distance_CPT_Presence_Produit := 520, [19].Comas.Consigne_Vitesse_Manu_Tour := 10.0, [19].Comas.Consigne_Acc_Decc_Manu_Tour := 10.0, [19].Comas.Mode_Decoreuse_Cam_Logique := 1, [19].Comas.Reserve_Real6 := 200.0, [20].Name := 'SAB CHOCO 314SAB005', [20].Comas.Pas_Machine := 75, [20].Comas.Came_Maitre[1].Master := 75.0, [20].Comas.Came_Maitre[1].Slave := 75.0, [20].Comas.Longueur_Came_Maitre := 2, [20].Comas.Tete.Stop_Cam_Logique_Degagement := 10.0, [20].Comas.Tete.Position_Degagement_H := 50.0, [20].Comas.Tete.Position_Degagement_V := 35.0, [20].Comas.Tete.Hauteur_Tete := -1, [20].Comas.Tete.Cam_Axe_Horizontal[1].Master := 1.0, [20].Comas.Tete.Cam_Axe_Horizontal[1].SegmentType := 1, [20].Comas.Tete.Cam_Axe_Horizontal[2].Master := 6.0, [20].Comas.Tete.Cam_Axe_Horizontal[2].Slave := 2.0, [20].Comas.Tete.Cam_Axe_Horizontal[3].Master := 36.0, [20].Comas.Tete.Cam_Axe_Horizontal[3].Slave := 37.0, [20].Comas.Tete.Cam_Axe_Horizontal[3].SegmentType := 1, [20].Comas.Tete.Cam_Axe_Horizontal[4].Master := 46.0, [20].Comas.Tete.Cam_Axe_Horizontal[4].Slave := 42.0, [20].Comas.Tete.Cam_Axe_Horizontal[5].Master := 51.0, [20].Comas.Tete.Cam_Axe_Horizontal[5].Slave := 42.0, [20].Comas.Tete.Cam_Axe_Horizontal[5].SegmentType := 1, [20].Comas.Tete.Cam_Axe_Horizontal[6].Master := 61.0, [20].Comas.Tete.Cam_Axe_Horizontal[6].Slave := 32.0, [20].Comas.Tete.Cam_Axe_Horizontal[6].SegmentType := 1, [20].Comas.Tete.Cam_Axe_Horizontal[7].Master := 75.0, [20].Comas.Tete.Cam_Axe_Vertical[1].Master := 1.0, [20].Comas.Tete.Cam_Axe_Vertical[2].Master := 6.0, [20].Comas.Tete.Cam_Axe_Vertical[3].Master := 26.0, [20].Comas.Tete.Cam_Axe_Vertical[3].SegmentType := 1, [20].Comas.Tete.Cam_Axe_Vertical[4].Master := 36.0, [20].Comas.Tete.Cam_Axe_Vertical[4].Slave := 10.0, [20].Comas.Tete.Cam_Axe_Vertical[5].Master := 64.0, [20].Comas.Tete.Cam_Axe_Vertical[5].Slave := 10.0, [20].Comas.Tete.Cam_Axe_Vertical[5].SegmentType := 1, [20].Comas.Tete.Cam_Axe_Vertical[6].Master := 74.0, [20].Comas.Tete.Cam_Axe_Vertical[7].Master := 75.0, [20].Comas.Tete.Longueur_Cam_Axe_H := 8, [20].Comas.Tete.Offset_Vertical_Gauche := 38.0, [20].Comas.Tete.Offset_Horizontal_Gauche := 95.0,
        [20].Comas.Tete.Cam_Axe_Horizontal_Pan.B.x := 1.0, [20].Comas.Tete.Cam_Axe_Horizontal_Pan.C.x := 5.0, [20].Comas.Tete.Cam_Axe_Horizontal_Pan.C.y := 2.0, [20].Comas.Tete.Cam_Axe_Horizontal_Pan.D.x := 30.0, [20].Comas.Tete.Cam_Axe_Horizontal_Pan.D.y := 30.0, [20].Comas.Tete.Cam_Axe_Horizontal_Pan.E.x := 10.0, [20].Comas.Tete.Cam_Axe_Horizontal_Pan.E.y := 5.0, [20].Comas.Tete.Cam_Axe_Horizontal_Pan.F.x := 5.0, [20].Comas.Tete.Cam_Axe_Horizontal_Pan.G.x := 10.0, [20].Comas.Tete.Cam_Axe_Horizontal_Pan.G.y := -10.0, [20].Comas.Tete.Cam_Axe_Vertical_Pan.K.x := -10.0, [20].Comas.Tete.Cam_Axe_Vertical_Pan.L.x := -10.0, [20].Comas.Tete.Cam_Axe_Vertical_Pan.L.y := 10.0, [20].Comas.Tete.Cam_Axe_Vertical_Pan.M.x := 13.0, [20].Comas.Tete.Cam_Axe_Vertical_Pan.M.y := 10.0, [20].Comas.Tete.Cam_Axe_Vertical_Pan.N.x := 13.0, [20].Comas.Tete.Offset_Vertical_Droit := 45.0, [20].Comas.Tete.Offset_Horizontal_Droit := 95.0, [20].Comas.Tete.Reserve_Real1 := 5.0, [20].Comas.Pompe.Start_Cam_Logique_Avance := -9.0, [20].Comas.Pompe.Stop_Cam_Logique_Avance := 11.0, [20].Comas.Pompe.Start_Cam_Logique_Recul := 11.0, [20].Comas.Pompe.Stop_Cam_Logique_Recul := 23.5, [20].Comas.Pompe.Consigne_Vitesse_Avance := 34.0, [20].Comas.Pompe.Consigne_Acc_Dec_Avance := 40.0, [20].Comas.Pompe.Consigne_Jerk_Avance := 100.0, [20].Comas.Pompe.Consigne_Vitesse_Recul := -31.0, [20].Comas.Pompe.Consigne_Acc_Dec_Recul := 40.0, [20].Comas.Pompe.Consigne_Jerk_Recul := 100.0, [20].Comas.Pompe.Points_Pan.O.x := -15.0, [20].Comas.Pompe.Points_Pan.Q.x := 20.0, [20].Comas.Pompe.Points_Pan.S.x := -15.0, [20].Comas.Pompe.Points_Pan.U.x := 12.5, [20].Comas.Pompe.Reserve_Bool1 := 1, [20].Comas.Rouleaux.Consigne_Vitesse := 25.0, [20].Comas.Rouleaux.Consigne_Acc_Dec := 40.0, [20].Comas.Rouleaux.Consigne_Jerk := 100.0, [20].Comas.Coupe_Fil.Start_Cam_Logique_Virtuelle := 11.0, [20].Comas.Coupe_Fil.Stop_Cam_Logique_Virtuelle := 21.0, [20].Comas.Coupe_Fil.Consigne_Vitesse_Virtuelle := 200.0, [20].Comas.Coupe_Fil.Consigne_Acc_Dec_Virtuelle := 1000.0, [20].Comas.Coupe_Fil.Consigne_Jerk_Virtuelle := 50.0, [20].Comas.Coupe_Fil.Cam_Axe[0].SegmentType := 1, [20].Comas.Coupe_Fil.Cam_Axe[1].Master := 180.0, [20].Comas.Coupe_Fil.Cam_Axe[1].Slave := 90.0, [20].Comas.Coupe_Fil.Cam_Axe[2].Master := 360.0, [20].Comas.Coupe_Fil.Cam_Axe[2].Slave := 360.0, [20].Comas.Coupe_Fil.Cam_Axe[2].SegmentType := 1, [20].Comas.Coupe_Fil.Points_Pan.W.x := 30.0, [20].Comas.Consigne_Vitesse_Manu_mm := 4.0, [20].Comas.Consigne_Acc_Decc_Manu_mm := 10.0, [20].Comas.Consigne_Jerk_Manu := 100.0, [20].Comas.Activation_Cam_Auto := 1, [20].Comas.Distance_CPT_Presence_Produit := 520, [20].Comas.Consigne_Vitesse_Manu_Tour := 10.0, [20].Comas.Consigne_Acc_Decc_Manu_Tour := 10.0, [20].Comas.Mode_Decoreuse_Cam_Logique := 1, [20].Comas.Reserve_Real6 := 200.0, [21].Name := 'TUIL COCO 311PBL006', [21].Comas.Pas_Machine := 60,
        [21].Comas.Came_Maitre[1].Master := 60.0, [21].Comas.Came_Maitre[1].Slave := 60.0, [21].Comas.Longueur_Came_Maitre := 2, [21].Comas.Tete.Stop_Cam_Logique_Degagement := 10.0, [21].Comas.Tete.Position_Degagement_H := 50.0, [21].Comas.Tete.Position_Degagement_V := 35.0, [21].Comas.Tete.Hauteur_Tete := -1, [21].Comas.Tete.Cam_Axe_Horizontal[1].Master := 1.0, [21].Comas.Tete.Cam_Axe_Horizontal[1].SegmentType := 1, [21].Comas.Tete.Cam_Axe_Horizontal[2].Master := 6.0, [21].Comas.Tete.Cam_Axe_Horizontal[2].Slave := 2.0, [21].Comas.Tete.Cam_Axe_Horizontal[3].Master := 21.0, [21].Comas.Tete.Cam_Axe_Horizontal[3].Slave := 27.0, [21].Comas.Tete.Cam_Axe_Horizontal[3].SegmentType := 1, [21].Comas.Tete.Cam_Axe_Horizontal[4].Master := 31.0, [21].Comas.Tete.Cam_Axe_Horizontal[4].Slave := 32.0, [21].Comas.Tete.Cam_Axe_Horizontal[5].Master := 36.0, [21].Comas.Tete.Cam_Axe_Horizontal[5].Slave := 32.0, [21].Comas.Tete.Cam_Axe_Horizontal[5].SegmentType := 1, [21].Comas.Tete.Cam_Axe_Horizontal[6].Master := 46.0, [21].Comas.Tete.Cam_Axe_Horizontal[6].Slave := 22.0, [21].Comas.Tete.Cam_Axe_Horizontal[6].SegmentType := 1, [21].Comas.Tete.Cam_Axe_Horizontal[7].Master := 60.0, [21].Comas.Tete.Cam_Axe_Vertical[1].Master := 1.0, [21].Comas.Tete.Cam_Axe_Vertical[2].Master := 6.0, [21].Comas.Tete.Cam_Axe_Vertical[3].Master := 11.0, [21].Comas.Tete.Cam_Axe_Vertical[3].SegmentType := 1, [21].Comas.Tete.Cam_Axe_Vertical[4].Master := 21.0, [21].Comas.Tete.Cam_Axe_Vertical[4].Slave := 3.0, [21].Comas.Tete.Cam_Axe_Vertical[5].Master := 41.0, [21].Comas.Tete.Cam_Axe_Vertical[5].Slave := 3.0, [21].Comas.Tete.Cam_Axe_Vertical[5].SegmentType := 1, [21].Comas.Tete.Cam_Axe_Vertical[6].Master := 56.0, [21].Comas.Tete.Cam_Axe_Vertical[7].Master := 60.0, [21].Comas.Tete.Longueur_Cam_Axe_H := 8, [21].Comas.Tete.Offset_Vertical_Gauche := 38.0, [21].Comas.Tete.Offset_Horizontal_Gauche := 95.0, [21].Comas.Tete.Cam_Axe_Horizontal_Pan.B.x := 1.0, [21].Comas.Tete.Cam_Axe_Horizontal_Pan.C.x := 5.0, [21].Comas.Tete.Cam_Axe_Horizontal_Pan.C.y := 2.0, [21].Comas.Tete.Cam_Axe_Horizontal_Pan.D.x := 15.0, [21].Comas.Tete.Cam_Axe_Horizontal_Pan.D.y := 25.0, [21].Comas.Tete.Cam_Axe_Horizontal_Pan.E.x := 10.0, [21].Comas.Tete.Cam_Axe_Horizontal_Pan.E.y := 5.0, [21].Comas.Tete.Cam_Axe_Horizontal_Pan.F.x := 5.0, [21].Comas.Tete.Cam_Axe_Horizontal_Pan.G.x := 10.0, [21].Comas.Tete.Cam_Axe_Horizontal_Pan.G.y := -10.0, [21].Comas.Tete.Cam_Axe_Vertical_Pan.K.x := -10.0, [21].Comas.Tete.Cam_Axe_Vertical_Pan.L.x := -10.0, [21].Comas.Tete.Cam_Axe_Vertical_Pan.L.y := 3.0, [21].Comas.Tete.Cam_Axe_Vertical_Pan.M.x := 5.0, [21].Comas.Tete.Cam_Axe_Vertical_Pan.M.y := 3.0, [21].Comas.Tete.Cam_Axe_Vertical_Pan.N.x := 10.0, [21].Comas.Tete.Offset_Vertical_Droit := 45.0, [21].Comas.Tete.Offset_Horizontal_Droit := 95.0, [21].Comas.Pompe.Start_Cam_Logique_Avance := -8.0, [21].Comas.Pompe.Stop_Cam_Logique_Avance := 7.0, [21].Comas.Pompe.Start_Cam_Logique_Recul := 7.0, [21].Comas.Pompe.Stop_Cam_Logique_Recul := 22.0, [21].Comas.Pompe.Consigne_Vitesse_Avance := 42.8,
        [21].Comas.Pompe.Consigne_Acc_Dec_Avance := 40.0, [21].Comas.Pompe.Consigne_Jerk_Avance := 100.0, [21].Comas.Pompe.Consigne_Vitesse_Recul := -28.0, [21].Comas.Pompe.Consigne_Acc_Dec_Recul := 40.0, [21].Comas.Pompe.Consigne_Jerk_Recul := 100.0, [21].Comas.Pompe.Points_Pan.O.x := -14.0, [21].Comas.Pompe.Points_Pan.Q.x := 15.0, [21].Comas.Pompe.Points_Pan.S.x := -4.0, [21].Comas.Pompe.Points_Pan.U.x := 15.0, [21].Comas.Pompe.Reserve_Bool1 := 1, [21].Comas.Rouleaux.Consigne_Vitesse := 25.0, [21].Comas.Rouleaux.Consigne_Acc_Dec := 40.0, [21].Comas.Rouleaux.Consigne_Jerk := 100.0, [21].Comas.Rouleaux.Reserve_Real1 := -15.0, [21].Comas.Coupe_Fil.Start_Cam_Logique_Virtuelle := 11.0, [21].Comas.Coupe_Fil.Stop_Cam_Logique_Virtuelle := 21.0, [21].Comas.Coupe_Fil.Consigne_Vitesse_Virtuelle := 200.0, [21].Comas.Coupe_Fil.Consigne_Acc_Dec_Virtuelle := 1000.0, [21].Comas.Coupe_Fil.Consigne_Jerk_Virtuelle := 50.0, [21].Comas.Coupe_Fil.Cam_Axe[0].SegmentType := 1, [21].Comas.Coupe_Fil.Cam_Axe[1].Master := 180.0, [21].Comas.Coupe_Fil.Cam_Axe[1].Slave := 90.0, [21].Comas.Coupe_Fil.Cam_Axe[2].Master := 360.0, [21].Comas.Coupe_Fil.Cam_Axe[2].Slave := 360.0, [21].Comas.Coupe_Fil.Cam_Axe[2].SegmentType := 1, [21].Comas.Coupe_Fil.Points_Pan.W.x := 30.0, [21].Comas.Consigne_Vitesse_Manu_mm := 4.0, [21].Comas.Consigne_Acc_Decc_Manu_mm := 10.0, [21].Comas.Consigne_Jerk_Manu := 100.0, [21].Comas.Activation_Cam_Auto := 1, [21].Comas.Distance_CPT_Presence_Produit := 520, [21].Comas.Consigne_Vitesse_Manu_Tour := 10.0, [21].Comas.Consigne_Acc_Decc_Manu_Tour := 10.0, [21].Comas.Mode_Decoreuse_Cam_Logique := 1, [21].Comas.Reserve_Real6 := 200.0, [22].Name := 'TARTELETTE 100', [22].Comas.Pas_Machine := 110, [22].Comas.Came_Maitre[1].Master := 110.0, [22].Comas.Came_Maitre[1].Slave := 110.0, [22].Comas.Longueur_Came_Maitre := 2, [22].Comas.Tete.Stop_Cam_Logique_Degagement := 10.0, [22].Comas.Tete.Position_Degagement_H := 50.0, [22].Comas.Tete.Position_Degagement_V := 35.0, [22].Comas.Tete.Cam_Axe_Horizontal[1].Master := 1.0, [22].Comas.Tete.Cam_Axe_Horizontal[1].SegmentType := 1, [22].Comas.Tete.Cam_Axe_Horizontal[2].Master := 6.0, [22].Comas.Tete.Cam_Axe_Horizontal[2].Slave := 5.0, [22].Comas.Tete.Cam_Axe_Horizontal[3].Master := 36.0, [22].Comas.Tete.Cam_Axe_Horizontal[3].Slave := 50.0, [22].Comas.Tete.Cam_Axe_Horizontal[3].SegmentType := 1, [22].Comas.Tete.Cam_Axe_Horizontal[4].Master := 46.0, [22].Comas.Tete.Cam_Axe_Horizontal[4].Slave := 60.0, [22].Comas.Tete.Cam_Axe_Horizontal[5].Master := 56.0, [22].Comas.Tete.Cam_Axe_Horizontal[5].Slave := 60.0, [22].Comas.Tete.Cam_Axe_Horizontal[5].SegmentType := 1, [22].Comas.Tete.Cam_Axe_Horizontal[6].Master := 66.0, [22].Comas.Tete.Cam_Axe_Horizontal[6].Slave := 55.0, [22].Comas.Tete.Cam_Axe_Horizontal[6].SegmentType := 1, [22].Comas.Tete.Cam_Axe_Horizontal[7].Master := 110.0, [22].Comas.Tete.Cam_Axe_Vertical[1].Master := 1.0,
        [22].Comas.Tete.Cam_Axe_Vertical[2].Master := 6.0, [22].Comas.Tete.Cam_Axe_Vertical[2].Slave := -3.0, [22].Comas.Tete.Cam_Axe_Vertical[3].Master := 26.0, [22].Comas.Tete.Cam_Axe_Vertical[3].Slave := -5.0, [22].Comas.Tete.Cam_Axe_Vertical[3].SegmentType := 1, [22].Comas.Tete.Cam_Axe_Vertical[4].Master := 36.0, [22].Comas.Tete.Cam_Axe_Vertical[4].Slave := -3.0, [22].Comas.Tete.Cam_Axe_Vertical[5].Master := 86.0, [22].Comas.Tete.Cam_Axe_Vertical[5].Slave := 22.0, [22].Comas.Tete.Cam_Axe_Vertical[5].SegmentType := 1, [22].Comas.Tete.Cam_Axe_Vertical[6].Master := 104.0, [22].Comas.Tete.Cam_Axe_Vertical[7].Master := 110.0, [22].Comas.Tete.Longueur_Cam_Axe_H := 8, [22].Comas.Tete.Offset_Vertical_Gauche := 38.0, [22].Comas.Tete.Offset_Horizontal_Gauche := 95.0, [22].Comas.Tete.Cam_Axe_Horizontal_Pan.B.x := 1.0, [22].Comas.Tete.Cam_Axe_Horizontal_Pan.C.x := 5.0, [22].Comas.Tete.Cam_Axe_Horizontal_Pan.C.y := 5.0, [22].Comas.Tete.Cam_Axe_Horizontal_Pan.D.x := 30.0, [22].Comas.Tete.Cam_Axe_Horizontal_Pan.D.y := 45.0, [22].Comas.Tete.Cam_Axe_Horizontal_Pan.E.x := 10.0, [22].Comas.Tete.Cam_Axe_Horizontal_Pan.E.y := 10.0, [22].Comas.Tete.Cam_Axe_Horizontal_Pan.F.x := 10.0, [22].Comas.Tete.Cam_Axe_Horizontal_Pan.G.x := 10.0, [22].Comas.Tete.Cam_Axe_Horizontal_Pan.G.y := -5.0, [22].Comas.Tete.Cam_Axe_Vertical_Pan.J.y := -3.0, [22].Comas.Tete.Cam_Axe_Vertical_Pan.K.x := -10.0, [22].Comas.Tete.Cam_Axe_Vertical_Pan.K.y := -5.0, [22].Comas.Tete.Cam_Axe_Vertical_Pan.L.x := -10.0, [22].Comas.Tete.Cam_Axe_Vertical_Pan.L.y := -3.0, [22].Comas.Tete.Cam_Axe_Vertical_Pan.M.x := 30.0, [22].Comas.Tete.Cam_Axe_Vertical_Pan.M.y := 22.0, [22].Comas.Tete.Cam_Axe_Vertical_Pan.N.x := 38.0, [22].Comas.Tete.Offset_Vertical_Droit := 45.0, [22].Comas.Tete.Offset_Horizontal_Droit := 95.0, [22].Comas.Pompe.Start_Cam_Logique_Avance := -9.0, [22].Comas.Pompe.Stop_Cam_Logique_Avance := 11.0, [22].Comas.Pompe.Start_Cam_Logique_Recul := 21.0, [22].Comas.Pompe.Stop_Cam_Logique_Recul := 36.0, [22].Comas.Pompe.Consigne_Vitesse_Avance := 17.5, [22].Comas.Pompe.Consigne_Acc_Dec_Avance := 40.0, [22].Comas.Pompe.Consigne_Jerk_Avance := 100.0, [22].Comas.Pompe.Consigne_Vitesse_Recul := -19.5, [22].Comas.Pompe.Consigne_Acc_Dec_Recul := 40.0, [22].Comas.Pompe.Consigne_Jerk_Recul := 100.0, [22].Comas.Pompe.Points_Pan.O.x := -15.0, [22].Comas.Pompe.Points_Pan.Q.x := 20.0, [22].Comas.Pompe.Points_Pan.S.x := -5.0, [22].Comas.Pompe.Points_Pan.U.x := 15.0, [22].Comas.Pompe.Reserve_Bool1 := 1, [22].Comas.Rouleaux.Consigne_Vitesse := 5.0, [22].Comas.Rouleaux.Consigne_Acc_Dec := 40.0, [22].Comas.Rouleaux.Consigne_Jerk := 100.0, [22].Comas.Rouleaux.Reserve_Real1 := -10.0, [22].Comas.Coupe_Fil.Start_Cam_Logique_Virtuelle := 11.0, [22].Comas.Coupe_Fil.Stop_Cam_Logique_Virtuelle := 21.0, [22].Comas.Coupe_Fil.Consigne_Vitesse_Virtuelle := 200.0, [22].Comas.Coupe_Fil.Consigne_Acc_Dec_Virtuelle := 1000.0, [22].Comas.Coupe_Fil.Consigne_Jerk_Virtuelle := 50.0, [22].Comas.Coupe_Fil.Cam_Axe[0].SegmentType := 1,
        [22].Comas.Coupe_Fil.Cam_Axe[1].Master := 180.0, [22].Comas.Coupe_Fil.Cam_Axe[1].Slave := 90.0, [22].Comas.Coupe_Fil.Cam_Axe[2].Master := 360.0, [22].Comas.Coupe_Fil.Cam_Axe[2].Slave := 360.0, [22].Comas.Coupe_Fil.Cam_Axe[2].SegmentType := 1, [22].Comas.Coupe_Fil.Points_Pan.W.x := 30.0, [22].Comas.Consigne_Vitesse_Manu_mm := 2.0, [22].Comas.Consigne_Acc_Decc_Manu_mm := 10.0, [22].Comas.Consigne_Jerk_Manu := 100.0, [22].Comas.Activation_Cam_Auto := 1, [22].Comas.Mode_CPT_Presence := 1, [22].Comas.Distance_CPT_Presence_Produit := 575, [22].Comas.Consigne_Vitesse_Manu_Tour := 10.0, [22].Comas.Consigne_Acc_Decc_Manu_Tour := 10.0, [22].Comas.Reserve_Real1 := 25.0, [22].Comas.Reserve_Real2 := 10.0, [22].Comas.Reserve_Real3 := 1.0, [22].Comas.Reserve_Real4 := 1.0, [22].Comas.Reserve_Real5 := 5.0, [22].Comas.Reserve_Real6 := 200.0, [22].Reserve_Real2 := 200.0, [22].Reserve_Real3 := 10.0, [22].Reserve_Bool4 := 1, [23].Name := 'SAB CACAO SSP', [23].Comas.Pas_Machine := 75, [23].Comas.Came_Maitre[1].Master := 75.0, [23].Comas.Came_Maitre[1].Slave := 75.0, [23].Comas.Longueur_Came_Maitre := 2, [23].Comas.Tete.Stop_Cam_Logique_Degagement := 10.0, [23].Comas.Tete.Position_Degagement_H := 50.0, [23].Comas.Tete.Position_Degagement_V := 35.0, [23].Comas.Tete.Hauteur_Tete := -5, [23].Comas.Tete.Cam_Axe_Horizontal[1].Master := 1.0, [23].Comas.Tete.Cam_Axe_Horizontal[1].SegmentType := 1, [23].Comas.Tete.Cam_Axe_Horizontal[2].Master := 6.0, [23].Comas.Tete.Cam_Axe_Horizontal[2].Slave := 7.0, [23].Comas.Tete.Cam_Axe_Horizontal[2].SegmentType := 1, [23].Comas.Tete.Cam_Axe_Horizontal[3].Master := 36.0, [23].Comas.Tete.Cam_Axe_Horizontal[3].Slave := 42.0, [23].Comas.Tete.Cam_Axe_Horizontal[3].SegmentType := 1, [23].Comas.Tete.Cam_Axe_Horizontal[4].Master := 46.0, [23].Comas.Tete.Cam_Axe_Horizontal[4].Slave := 47.0, [23].Comas.Tete.Cam_Axe_Horizontal[5].Master := 51.0, [23].Comas.Tete.Cam_Axe_Horizontal[5].Slave := 47.0, [23].Comas.Tete.Cam_Axe_Horizontal[5].SegmentType := 1, [23].Comas.Tete.Cam_Axe_Horizontal[6].Master := 61.0, [23].Comas.Tete.Cam_Axe_Horizontal[6].Slave := 37.0, [23].Comas.Tete.Cam_Axe_Horizontal[6].SegmentType := 1, [23].Comas.Tete.Cam_Axe_Horizontal[7].Master := 75.0, [23].Comas.Tete.Cam_Axe_Vertical[1].Master := 1.0, [23].Comas.Tete.Cam_Axe_Vertical[2].Master := 6.0, [23].Comas.Tete.Cam_Axe_Vertical[3].Master := 26.0, [23].Comas.Tete.Cam_Axe_Vertical[3].SegmentType := 1, [23].Comas.Tete.Cam_Axe_Vertical[4].Master := 36.0, [23].Comas.Tete.Cam_Axe_Vertical[4].Slave := 22.0, [23].Comas.Tete.Cam_Axe_Vertical[5].Master := 64.0, [23].Comas.Tete.Cam_Axe_Vertical[5].Slave := 22.0, [23].Comas.Tete.Cam_Axe_Vertical[5].SegmentType := 1, [23].Comas.Tete.Cam_Axe_Vertical[6].Master := 74.0, [23].Comas.Tete.Cam_Axe_Vertical[7].Master := 75.0,
        [23].Comas.Tete.Longueur_Cam_Axe_H := 8, [23].Comas.Tete.Offset_Vertical_Gauche := 38.0, [23].Comas.Tete.Offset_Horizontal_Gauche := 95.0, [23].Comas.Tete.Cam_Axe_Horizontal_Pan.B.x := 1.0, [23].Comas.Tete.Cam_Axe_Horizontal_Pan.C.x := 5.0, [23].Comas.Tete.Cam_Axe_Horizontal_Pan.C.y := 7.0, [23].Comas.Tete.Cam_Axe_Horizontal_Pan.D.x := 30.0, [23].Comas.Tete.Cam_Axe_Horizontal_Pan.D.y := 30.0, [23].Comas.Tete.Cam_Axe_Horizontal_Pan.E.x := 10.0, [23].Comas.Tete.Cam_Axe_Horizontal_Pan.E.y := 5.0, [23].Comas.Tete.Cam_Axe_Horizontal_Pan.F.x := 5.0, [23].Comas.Tete.Cam_Axe_Horizontal_Pan.G.x := 10.0, [23].Comas.Tete.Cam_Axe_Horizontal_Pan.G.y := -10.0, [23].Comas.Tete.Cam_Axe_Vertical_Pan.K.x := -10.0, [23].Comas.Tete.Cam_Axe_Vertical_Pan.L.x := -10.0, [23].Comas.Tete.Cam_Axe_Vertical_Pan.L.y := 22.0, [23].Comas.Tete.Cam_Axe_Vertical_Pan.M.x := 13.0, [23].Comas.Tete.Cam_Axe_Vertical_Pan.M.y := 22.0, [23].Comas.Tete.Cam_Axe_Vertical_Pan.N.x := 13.0, [23].Comas.Tete.Offset_Vertical_Droit := 45.0, [23].Comas.Tete.Offset_Horizontal_Droit := 95.0, [23].Comas.Tete.Reserve_Real1 := 5.0, [23].Comas.Pompe.Start_Cam_Logique_Avance := -9.0, [23].Comas.Pompe.Stop_Cam_Logique_Avance := 11.0, [23].Comas.Pompe.Start_Cam_Logique_Recul := 11.0, [23].Comas.Pompe.Stop_Cam_Logique_Recul := 23.5, [23].Comas.Pompe.Consigne_Vitesse_Avance := 40.8, [23].Comas.Pompe.Consigne_Acc_Dec_Avance := 40.0, [23].Comas.Pompe.Consigne_Jerk_Avance := 100.0, [23].Comas.Pompe.Consigne_Vitesse_Recul := -34.0, [23].Comas.Pompe.Consigne_Acc_Dec_Recul := 40.0, [23].Comas.Pompe.Consigne_Jerk_Recul := 100.0, [23].Comas.Pompe.Points_Pan.O.x := -15.0, [23].Comas.Pompe.Points_Pan.Q.x := 20.0, [23].Comas.Pompe.Points_Pan.S.x := -15.0, [23].Comas.Pompe.Points_Pan.U.x := 12.5, [23].Comas.Pompe.Reserve_Bool1 := 1, [23].Comas.Rouleaux.Consigne_Vitesse := 21.0, [23].Comas.Rouleaux.Consigne_Acc_Dec := 40.0, [23].Comas.Rouleaux.Consigne_Jerk := 100.0, [23].Comas.Coupe_Fil.Start_Cam_Logique_Virtuelle := 11.0, [23].Comas.Coupe_Fil.Stop_Cam_Logique_Virtuelle := 21.0, [23].Comas.Coupe_Fil.Consigne_Vitesse_Virtuelle := 200.0, [23].Comas.Coupe_Fil.Consigne_Acc_Dec_Virtuelle := 1000.0, [23].Comas.Coupe_Fil.Consigne_Jerk_Virtuelle := 50.0, [23].Comas.Coupe_Fil.Cam_Axe[0].SegmentType := 1, [23].Comas.Coupe_Fil.Cam_Axe[1].Master := 180.0, [23].Comas.Coupe_Fil.Cam_Axe[1].Slave := 90.0, [23].Comas.Coupe_Fil.Cam_Axe[2].Master := 360.0, [23].Comas.Coupe_Fil.Cam_Axe[2].Slave := 360.0, [23].Comas.Coupe_Fil.Cam_Axe[2].SegmentType := 1, [23].Comas.Coupe_Fil.Points_Pan.W.x := 30.0, [23].Comas.Consigne_Vitesse_Manu_mm := 4.0, [23].Comas.Consigne_Acc_Decc_Manu_mm := 10.0, [23].Comas.Consigne_Jerk_Manu := 100.0, [23].Comas.Activation_Cam_Auto := 1, [23].Comas.Distance_CPT_Presence_Produit := 520, [23].Comas.Consigne_Vitesse_Manu_Tour := 10.0, [23].Comas.Consigne_Acc_Decc_Manu_Tour := 10.0, [23].Comas.Mode_Decoreuse_Cam_Logique := 1,
        [23].Comas.Reserve_Real3 := 1.0, [23].Comas.Reserve_Real4 := 1.0, [23].Comas.Reserve_Real5 := 5.0, [23].Comas.Reserve_Real6 := 200.0, [23].Reserve_Real2 := 200.0, [23].Reserve_Real3 := 10.0, [24].Name := 'Palet citron MDLZ', [24].Comas.Pas_Machine := 70, [24].Comas.Came_Maitre[1].Master := 70.0, [24].Comas.Came_Maitre[1].Slave := 70.0, [24].Comas.Longueur_Came_Maitre := 2, [24].Comas.Tete.Stop_Cam_Logique_Degagement := 10.0, [24].Comas.Tete.Position_Degagement_H := 50.0, [24].Comas.Tete.Position_Degagement_V := 35.0, [24].Comas.Tete.Hauteur_Tete := -2, [24].Comas.Tete.Cam_Axe_Horizontal[1].Master := 1.0, [24].Comas.Tete.Cam_Axe_Horizontal[1].SegmentType := 1, [24].Comas.Tete.Cam_Axe_Horizontal[2].Master := 6.0, [24].Comas.Tete.Cam_Axe_Horizontal[2].Slave := 2.0, [24].Comas.Tete.Cam_Axe_Horizontal[3].Master := 31.0, [24].Comas.Tete.Cam_Axe_Horizontal[3].Slave := 32.0, [24].Comas.Tete.Cam_Axe_Horizontal[3].SegmentType := 1, [24].Comas.Tete.Cam_Axe_Horizontal[4].Master := 41.0, [24].Comas.Tete.Cam_Axe_Horizontal[4].Slave := 42.0, [24].Comas.Tete.Cam_Axe_Horizontal[5].Master := 46.0, [24].Comas.Tete.Cam_Axe_Horizontal[5].Slave := 42.0, [24].Comas.Tete.Cam_Axe_Horizontal[5].SegmentType := 1, [24].Comas.Tete.Cam_Axe_Horizontal[6].Master := 56.0, [24].Comas.Tete.Cam_Axe_Horizontal[6].Slave := 32.0, [24].Comas.Tete.Cam_Axe_Horizontal[6].SegmentType := 1, [24].Comas.Tete.Cam_Axe_Horizontal[7].Master := 70.0, [24].Comas.Tete.Cam_Axe_Vertical[1].Master := 1.0, [24].Comas.Tete.Cam_Axe_Vertical[2].Master := 6.0, [24].Comas.Tete.Cam_Axe_Vertical[3].Master := 21.0, [24].Comas.Tete.Cam_Axe_Vertical[3].SegmentType := 1, [24].Comas.Tete.Cam_Axe_Vertical[4].Master := 31.0, [24].Comas.Tete.Cam_Axe_Vertical[4].Slave := 12.0, [24].Comas.Tete.Cam_Axe_Vertical[5].Master := 51.0, [24].Comas.Tete.Cam_Axe_Vertical[5].Slave := 5.0, [24].Comas.Tete.Cam_Axe_Vertical[5].SegmentType := 1, [24].Comas.Tete.Cam_Axe_Vertical[6].Master := 66.0, [24].Comas.Tete.Cam_Axe_Vertical[7].Master := 70.0, [24].Comas.Tete.Longueur_Cam_Axe_H := 8, [24].Comas.Tete.Offset_Vertical_Gauche := 38.0, [24].Comas.Tete.Offset_Horizontal_Gauche := 95.0, [24].Comas.Tete.Cam_Axe_Horizontal_Pan.B.x := 1.0, [24].Comas.Tete.Cam_Axe_Horizontal_Pan.C.x := 5.0, [24].Comas.Tete.Cam_Axe_Horizontal_Pan.C.y := 2.0, [24].Comas.Tete.Cam_Axe_Horizontal_Pan.D.x := 25.0, [24].Comas.Tete.Cam_Axe_Horizontal_Pan.D.y := 27.0, [24].Comas.Tete.Cam_Axe_Horizontal_Pan.E.x := 10.0, [24].Comas.Tete.Cam_Axe_Horizontal_Pan.E.y := 10.0, [24].Comas.Tete.Cam_Axe_Horizontal_Pan.F.x := 5.0, [24].Comas.Tete.Cam_Axe_Horizontal_Pan.G.x := 10.0, [24].Comas.Tete.Cam_Axe_Horizontal_Pan.G.y := -10.0, [24].Comas.Tete.Cam_Axe_Vertical_Pan.K.x := -10.0, [24].Comas.Tete.Cam_Axe_Vertical_Pan.L.x := -10.0, [24].Comas.Tete.Cam_Axe_Vertical_Pan.L.y := 12.0, [24].Comas.Tete.Cam_Axe_Vertical_Pan.M.x := 5.0, [24].Comas.Tete.Cam_Axe_Vertical_Pan.M.y := 5.0,
        [24].Comas.Tete.Cam_Axe_Vertical_Pan.N.x := 10.0, [24].Comas.Tete.Offset_Vertical_Droit := 45.0, [24].Comas.Tete.Offset_Horizontal_Droit := 95.0, [24].Comas.Tete.Reserve_Real1 := 3.0, [24].Comas.Pompe.Start_Cam_Logique_Avance := -9.0, [24].Comas.Pompe.Stop_Cam_Logique_Avance := 16.0, [24].Comas.Pompe.Start_Cam_Logique_Recul := 21.0, [24].Comas.Pompe.Stop_Cam_Logique_Recul := 33.0, [24].Comas.Pompe.Consigne_Vitesse_Avance := 19.4, [24].Comas.Pompe.Consigne_Acc_Dec_Avance := 40.0, [24].Comas.Pompe.Consigne_Jerk_Avance := 100.0, [24].Comas.Pompe.Consigne_Vitesse_Recul := -19.0, [24].Comas.Pompe.Consigne_Acc_Dec_Recul := 40.0, [24].Comas.Pompe.Consigne_Jerk_Recul := 100.0, [24].Comas.Pompe.Points_Pan.O.x := -15.0, [24].Comas.Pompe.Points_Pan.Q.x := 25.0, [24].Comas.Pompe.Points_Pan.U.x := 12.0, [24].Comas.Pompe.Reserve_Bool1 := 1, [24].Comas.Rouleaux.Syncho_Pompe := 1, [24].Comas.Rouleaux.Consigne_Vitesse := 20.0, [24].Comas.Rouleaux.Consigne_Acc_Dec := 40.0, [24].Comas.Rouleaux.Consigne_Jerk := 100.0, [24].Comas.Coupe_Fil.Start_Cam_Logique_Virtuelle := 11.0, [24].Comas.Coupe_Fil.Stop_Cam_Logique_Virtuelle := 21.0, [24].Comas.Coupe_Fil.Consigne_Vitesse_Virtuelle := 200.0, [24].Comas.Coupe_Fil.Consigne_Acc_Dec_Virtuelle := 1000.0, [24].Comas.Coupe_Fil.Consigne_Jerk_Virtuelle := 50.0, [24].Comas.Coupe_Fil.Cam_Axe[0].SegmentType := 1, [24].Comas.Coupe_Fil.Cam_Axe[1].Master := 180.0, [24].Comas.Coupe_Fil.Cam_Axe[1].Slave := 90.0, [24].Comas.Coupe_Fil.Cam_Axe[2].Master := 360.0, [24].Comas.Coupe_Fil.Cam_Axe[2].Slave := 360.0, [24].Comas.Coupe_Fil.Cam_Axe[2].SegmentType := 1, [24].Comas.Coupe_Fil.Points_Pan.W.x := 30.0, [24].Comas.Consigne_Vitesse_Manu_mm := 4.0, [24].Comas.Consigne_Acc_Decc_Manu_mm := 10.0, [24].Comas.Consigne_Jerk_Manu := 100.0, [24].Comas.Activation_Cam_Auto := 1, [24].Comas.Distance_CPT_Presence_Produit := 520, [24].Comas.Consigne_Vitesse_Manu_Tour := 10.0, [24].Comas.Consigne_Acc_Decc_Manu_Tour := 10.0, [24].Comas.Mode_Decoreuse_Cam_Logique := 1, [24].Comas.Reserve_Real3 := 1.0, [24].Comas.Reserve_Real4 := 1.0, [24].Comas.Reserve_Real5 := 5.0, [24].Comas.Reserve_Real6 := 200.0, [24].Reserve_Real2 := 200.0, [24].Reserve_Real3 := 10.0, [25].Name := 'Midoux MDLZ', [25].Comas.Pas_Machine := 60, [25].Comas.Came_Maitre[1].Master := 60.0, [25].Comas.Came_Maitre[1].Slave := 60.0, [25].Comas.Longueur_Came_Maitre := 2, [25].Comas.Tete.Stop_Cam_Logique_Degagement := 10.0, [25].Comas.Tete.Position_Degagement_H := 50.0, [25].Comas.Tete.Position_Degagement_V := 35.0, [25].Comas.Tete.Hauteur_Tete := -18, [25].Comas.Tete.Cam_Axe_Horizontal[1].Master := 1.0, [25].Comas.Tete.Cam_Axe_Horizontal[1].SegmentType := 1, [25].Comas.Tete.Cam_Axe_Horizontal[2].Master := 6.0,
        [25].Comas.Tete.Cam_Axe_Horizontal[2].Slave := 2.0, [25].Comas.Tete.Cam_Axe_Horizontal[3].Master := 21.0, [25].Comas.Tete.Cam_Axe_Horizontal[3].Slave := 27.0, [25].Comas.Tete.Cam_Axe_Horizontal[3].SegmentType := 1, [25].Comas.Tete.Cam_Axe_Horizontal[4].Master := 31.0, [25].Comas.Tete.Cam_Axe_Horizontal[4].Slave := 32.0, [25].Comas.Tete.Cam_Axe_Horizontal[5].Master := 36.0, [25].Comas.Tete.Cam_Axe_Horizontal[5].Slave := 32.0, [25].Comas.Tete.Cam_Axe_Horizontal[5].SegmentType := 1, [25].Comas.Tete.Cam_Axe_Horizontal[6].Master := 46.0, [25].Comas.Tete.Cam_Axe_Horizontal[6].Slave := 22.0, [25].Comas.Tete.Cam_Axe_Horizontal[6].SegmentType := 1, [25].Comas.Tete.Cam_Axe_Horizontal[7].Master := 60.0, [25].Comas.Tete.Cam_Axe_Vertical[1].Master := 1.0, [25].Comas.Tete.Cam_Axe_Vertical[2].Master := 6.0, [25].Comas.Tete.Cam_Axe_Vertical[3].Master := 11.0, [25].Comas.Tete.Cam_Axe_Vertical[3].SegmentType := 1, [25].Comas.Tete.Cam_Axe_Vertical[4].Master := 21.0, [25].Comas.Tete.Cam_Axe_Vertical[4].Slave := 3.0, [25].Comas.Tete.Cam_Axe_Vertical[5].Master := 41.0, [25].Comas.Tete.Cam_Axe_Vertical[5].Slave := 3.0, [25].Comas.Tete.Cam_Axe_Vertical[5].SegmentType := 1, [25].Comas.Tete.Cam_Axe_Vertical[6].Master := 56.0, [25].Comas.Tete.Cam_Axe_Vertical[7].Master := 60.0, [25].Comas.Tete.Longueur_Cam_Axe_H := 8, [25].Comas.Tete.Offset_Vertical_Gauche := 38.0, [25].Comas.Tete.Offset_Horizontal_Gauche := 95.0, [25].Comas.Tete.Cam_Axe_Horizontal_Pan.B.x := 1.0, [25].Comas.Tete.Cam_Axe_Horizontal_Pan.C.x := 5.0, [25].Comas.Tete.Cam_Axe_Horizontal_Pan.C.y := 2.0, [25].Comas.Tete.Cam_Axe_Horizontal_Pan.D.x := 15.0, [25].Comas.Tete.Cam_Axe_Horizontal_Pan.D.y := 25.0, [25].Comas.Tete.Cam_Axe_Horizontal_Pan.E.x := 10.0, [25].Comas.Tete.Cam_Axe_Horizontal_Pan.E.y := 5.0, [25].Comas.Tete.Cam_Axe_Horizontal_Pan.F.x := 5.0, [25].Comas.Tete.Cam_Axe_Horizontal_Pan.G.x := 10.0, [25].Comas.Tete.Cam_Axe_Horizontal_Pan.G.y := -10.0, [25].Comas.Tete.Cam_Axe_Vertical_Pan.K.x := -10.0, [25].Comas.Tete.Cam_Axe_Vertical_Pan.L.x := -10.0, [25].Comas.Tete.Cam_Axe_Vertical_Pan.L.y := 3.0, [25].Comas.Tete.Cam_Axe_Vertical_Pan.M.x := 5.0, [25].Comas.Tete.Cam_Axe_Vertical_Pan.M.y := 3.0, [25].Comas.Tete.Cam_Axe_Vertical_Pan.N.x := 10.0, [25].Comas.Tete.Offset_Vertical_Droit := 45.0, [25].Comas.Tete.Offset_Horizontal_Droit := 95.0, [25].Comas.Pompe.Start_Cam_Logique_Avance := -8.0, [25].Comas.Pompe.Stop_Cam_Logique_Avance := 7.0, [25].Comas.Pompe.Start_Cam_Logique_Recul := 7.0, [25].Comas.Pompe.Stop_Cam_Logique_Recul := 22.0, [25].Comas.Pompe.Consigne_Vitesse_Avance := 47.0, [25].Comas.Pompe.Consigne_Acc_Dec_Avance := 40.0, [25].Comas.Pompe.Consigne_Jerk_Avance := 100.0, [25].Comas.Pompe.Consigne_Vitesse_Recul := -28.0, [25].Comas.Pompe.Consigne_Acc_Dec_Recul := 40.0, [25].Comas.Pompe.Consigne_Jerk_Recul := 100.0, [25].Comas.Pompe.Points_Pan.O.x := -14.0, [25].Comas.Pompe.Points_Pan.Q.x := 15.0, [25].Comas.Pompe.Points_Pan.S.x := -4.0, [25].Comas.Pompe.Points_Pan.U.x := 15.0, [25].Comas.Pompe.Reserve_Bool1 := 1,
        [25].Comas.Rouleaux.Syncho_Pompe := 1, [25].Comas.Rouleaux.Consigne_Vitesse := 26.0, [25].Comas.Rouleaux.Consigne_Acc_Dec := 40.0, [25].Comas.Rouleaux.Consigne_Jerk := 100.0, [25].Comas.Rouleaux.Reserve_Real2 := 500.0, [25].Comas.Coupe_Fil.Start_Cam_Logique_Virtuelle := 11.0, [25].Comas.Coupe_Fil.Stop_Cam_Logique_Virtuelle := 21.0, [25].Comas.Coupe_Fil.Consigne_Vitesse_Virtuelle := 200.0, [25].Comas.Coupe_Fil.Consigne_Acc_Dec_Virtuelle := 1000.0, [25].Comas.Coupe_Fil.Consigne_Jerk_Virtuelle := 50.0, [25].Comas.Coupe_Fil.Cam_Axe[0].SegmentType := 1, [25].Comas.Coupe_Fil.Cam_Axe[1].Master := 180.0, [25].Comas.Coupe_Fil.Cam_Axe[1].Slave := 90.0, [25].Comas.Coupe_Fil.Cam_Axe[2].Master := 360.0, [25].Comas.Coupe_Fil.Cam_Axe[2].Slave := 360.0, [25].Comas.Coupe_Fil.Cam_Axe[2].SegmentType := 1, [25].Comas.Coupe_Fil.Points_Pan.W.x := 30.0, [25].Comas.Consigne_Vitesse_Manu_mm := 4.0, [25].Comas.Consigne_Acc_Decc_Manu_mm := 10.0, [25].Comas.Consigne_Jerk_Manu := 100.0, [25].Comas.Activation_Cam_Auto := 1, [25].Comas.Distance_CPT_Presence_Produit := 520, [25].Comas.Consigne_Vitesse_Manu_Tour := 10.0, [25].Comas.Consigne_Acc_Decc_Manu_Tour := 10.0, [25].Comas.Mode_Decoreuse_Cam_Logique := 1, [25].Comas.Reserve_Real3 := 1.0, [25].Comas.Reserve_Real4 := 1.0, [25].Comas.Reserve_Real5 := 5.0, [25].Comas.Reserve_Real6 := 200.0, [25].Reserve_Real2 := 200.0, [25].Reserve_Real3 := 10.0, [26].Name := 'HEKLA CONTINU', [26].Comas.Pas_Machine := 100, [26].Comas.Came_Maitre[1].Master := 100.0, [26].Comas.Came_Maitre[1].Slave := 100.0, [26].Comas.Longueur_Came_Maitre := 2, [26].Comas.Tete.Stop_Cam_Logique_Degagement := 10.0, [26].Comas.Tete.Position_Degagement_H := 50.0, [26].Comas.Tete.Position_Degagement_V := 35.0, [26].Comas.Tete.Hauteur_Tete := 26, [26].Comas.Tete.Cam_Axe_Horizontal[1].Master := 100.0, [26].Comas.Tete.Cam_Axe_Horizontal[3].SegmentType := 1, [26].Comas.Tete.Cam_Axe_Horizontal[5].SegmentType := 1, [26].Comas.Tete.Cam_Axe_Horizontal[6].SegmentType := 1, [26].Comas.Tete.Cam_Axe_Horizontal[7].Master := 100.0, [26].Comas.Tete.Cam_Axe_Vertical[1].Master := 100.0, [26].Comas.Tete.Cam_Axe_Vertical[3].SegmentType := 1, [26].Comas.Tete.Cam_Axe_Vertical[5].SegmentType := 1, [26].Comas.Tete.Cam_Axe_Vertical[7].Master := 100.0, [26].Comas.Tete.Longueur_Cam_Axe_H := 8, [26].Comas.Tete.Offset_Vertical_Gauche := 38.0, [26].Comas.Tete.Offset_Horizontal_Gauche := 95.0, [26].Comas.Tete.Offset_Vertical_Droit := 45.0, [26].Comas.Tete.Offset_Horizontal_Droit := 95.0, [26].Comas.Pompe.Stop_Cam_Logique_Avance := 100.0, [26].Comas.Pompe.Consigne_Vitesse_Avance := 3.5, [26].Comas.Pompe.Consigne_Acc_Dec_Avance := 40.0, [26].Comas.Pompe.Consigne_Jerk_Avance := 100.0, [26].Comas.Pompe.Consigne_Acc_Dec_Recul := 40.0, [26].Comas.Pompe.Consigne_Jerk_Recul := 100.0,
        [26].Comas.Rouleaux.Consigne_Vitesse := 25.0, [26].Comas.Rouleaux.Consigne_Acc_Dec := 40.0, [26].Comas.Rouleaux.Consigne_Jerk := 100.0, [26].Comas.Coupe_Fil.Start_Cam_Logique_Virtuelle := 11.0, [26].Comas.Coupe_Fil.Stop_Cam_Logique_Virtuelle := 21.0, [26].Comas.Coupe_Fil.Consigne_Vitesse_Virtuelle := 200.0, [26].Comas.Coupe_Fil.Consigne_Acc_Dec_Virtuelle := 1000.0, [26].Comas.Coupe_Fil.Consigne_Jerk_Virtuelle := 50.0, [26].Comas.Coupe_Fil.Cam_Axe[0].SegmentType := 1, [26].Comas.Coupe_Fil.Cam_Axe[1].Master := 180.0, [26].Comas.Coupe_Fil.Cam_Axe[1].Slave := 90.0, [26].Comas.Coupe_Fil.Cam_Axe[2].Master := 360.0, [26].Comas.Coupe_Fil.Cam_Axe[2].Slave := 360.0, [26].Comas.Coupe_Fil.Cam_Axe[2].SegmentType := 1, [26].Comas.Coupe_Fil.Points_Pan.W.x := 30.0, [26].Comas.Consigne_Vitesse_Manu_mm := 4.0, [26].Comas.Consigne_Acc_Decc_Manu_mm := 10.0, [26].Comas.Consigne_Jerk_Manu := 100.0, [26].Comas.Distance_CPT_Presence_Produit := 520, [26].Comas.Consigne_Vitesse_Manu_Tour := 10.0, [26].Comas.Consigne_Acc_Decc_Manu_Tour := 10.0, [26].Comas.Mode_Decoreuse_Cam_Logique := 1, [26].Comas.Reserve_Real3 := 1.0, [26].Comas.Reserve_Real4 := 1.0, [26].Comas.Reserve_Real5 := 5.0, [26].Comas.Reserve_Real6 := 200.0, [26].Reserve_Real2 := 200.0, [26].Reserve_Real3 := 10.0, [27].Name := 'Cookie 314MIN012', [27].Comas.Pas_Machine := 95, [27].Comas.Came_Maitre[1].Master := 95.0, [27].Comas.Came_Maitre[1].Slave := 95.0, [27].Comas.Longueur_Came_Maitre := 2, [27].Comas.Tete.Stop_Cam_Logique_Degagement := 10.0, [27].Comas.Tete.Position_Degagement_H := 50.0, [27].Comas.Tete.Position_Degagement_V := 35.0, [27].Comas.Tete.Hauteur_Tete := -8, [27].Comas.Tete.Cam_Axe_Horizontal[1].Master := 1.0, [27].Comas.Tete.Cam_Axe_Horizontal[1].SegmentType := 1, [27].Comas.Tete.Cam_Axe_Horizontal[2].Master := 11.0, [27].Comas.Tete.Cam_Axe_Horizontal[2].Slave := 5.0, [27].Comas.Tete.Cam_Axe_Horizontal[3].Master := 41.0, [27].Comas.Tete.Cam_Axe_Horizontal[3].Slave := 35.0, [27].Comas.Tete.Cam_Axe_Horizontal[3].SegmentType := 1, [27].Comas.Tete.Cam_Axe_Horizontal[4].Master := 51.0, [27].Comas.Tete.Cam_Axe_Horizontal[4].Slave := 40.0, [27].Comas.Tete.Cam_Axe_Horizontal[5].Master := 61.0, [27].Comas.Tete.Cam_Axe_Horizontal[5].Slave := 40.0, [27].Comas.Tete.Cam_Axe_Horizontal[5].SegmentType := 1, [27].Comas.Tete.Cam_Axe_Horizontal[6].Master := 71.0, [27].Comas.Tete.Cam_Axe_Horizontal[6].Slave := 30.0, [27].Comas.Tete.Cam_Axe_Horizontal[6].SegmentType := 1, [27].Comas.Tete.Cam_Axe_Horizontal[7].Master := 95.0, [27].Comas.Tete.Cam_Axe_Vertical[1].Master := 1.0, [27].Comas.Tete.Cam_Axe_Vertical[2].Master := 11.0, [27].Comas.Tete.Cam_Axe_Vertical[3].Master := 41.0, [27].Comas.Tete.Cam_Axe_Vertical[3].Slave := 2.0, [27].Comas.Tete.Cam_Axe_Vertical[3].SegmentType := 1, [27].Comas.Tete.Cam_Axe_Vertical[4].Master := 65.0, [27].Comas.Tete.Cam_Axe_Vertical[4].Slave := 15.0,
